Universal Robots PolyScope program: MAIN.urp

Program MAIN (installation=GD directory=/programs/GD createdIn=5.13.0 lastSavedIn=5.13.0 robotSerialNumber=20235201349)
Calibrated DH parameters: a=[0.000054, -0.419714, -0.551624, -0.000117, -0.00005, 0]; d=[0.180606, 361.576503, -382.621839, 21.219041, 0.119842, 0.115503]; alpha=[1.57022, -0.001233, 0.007049, 1.570107, -1.569424, 0]; deltaTheta=[0, -0.815667, 6.836137, 0.262718, -0.000001, 0]
InitVariablesNode
BeforeStart
  Script file /programs/GD/ROVI/ROVI_RESET.script
    | def ROVI_RESET():
    |   if (not socket_open(host,port,socket_name)):
    |     rovi_err=902
    |     return False
    |   end
    |   socket_send_line("X0()",socket_name)
    |   ret=socket_read_line(socket_name,socket_timeout)
    |   if (ret == "OK"):
    |     rovi_err=0
    |   elif (ret == "NG"):
    |     rovi_err=to_num(socket_read_line(socket_name,socket_timeout))
    |   else:
    |     ret="NG"
    |     rovi_err=903
    |   end
    |   socket_close(socket_name)
    |   if (rovi_err != 0):
    |     if (is_popup):
    |       popup(str_cat(ret,rovi_err),title="X0",warning=True,blocking=True)
    |     end
    |     return False
    |   else:
    |     return True
    |   end
    | end
  Script file /programs/GD/ROVI/ROVI_CAPTURE.script
    | def ROVI_CAPTURE():
    |   Y1=[0.0,0.0,0.0,0.0]
    | #  p=get_actual_tool_flange_pose()
    |   p=Bucket
    |   if (not socket_open(host,port,socket_name)):
    |     rovi_err=902
    |     return False
    |   end
    |   socket_send_string("X1(",socket_name)
    |   socket_send_string(p[0],socket_name)
    |   socket_send_string(",",socket_name)
    |   socket_send_string(p[1],socket_name)
    |   socket_send_string(",",socket_name)
    |   socket_send_string(p[2],socket_name)
    |   socket_send_string(",",socket_name)
    |   socket_send_string(p[3],socket_name)
    |   socket_send_string(",",socket_name)
    |   socket_send_string(p[4],socket_name)
    |   socket_send_string(",",socket_name)
    |   socket_send_string(p[5],socket_name)
    |   socket_send_line(")",socket_name)
    |   ret=socket_read_line(socket_name,socket_timeout)
    |   if (ret == "OK"):
    |     rovi_err=0
    |     f=socket_read_ascii_float(4,socket_name,socket_timeout)
    |     while (f[0]!=4):
    |       sleep(0.3)
    |       f=socket_read_ascii_float(4,socket_name,socket_timeout)
    |     end
    |     i=0
    |     while (i<4):
    |       Y1[i]=f[i+1]
    |       i=i+1
    |     end
    |   elif (ret == "NG"):
    |     rovi_err=to_num(socket_read_line(socket_name,socket_timeout))
    |   else:
    |     ret="NG"
    |     rovi_err=903
    |   end
    |   socket_close(socket_name)
    |   if (rovi_err != 0):
    |     if (is_popup):
    |       popup(str_cat(ret,rovi_err),title="X1",warning=True,blocking=True)
    |     end
    |     return False
    |   else:
    |     return True
    |   end
    | end
  Script file /programs/GD/ROVI/ROVI_SOLVE.script
    | def ROVI_SOLVE(is_popup=is_popup):
    |   buf=p[10000.0,0.0,0.0,0.0,0.0,0.0]
    |   if (not socket_open(host,port,socket_name)):
    |     rovi_err=902
    |     return False
    |   end
    |   socket_send_line("X2()",socket_name)
    |   ret=socket_read_line(socket_name,socket_timeout)
    |   if (ret == "OK"):
    |     rovi_err=0
    |     f=socket_read_ascii_float(6,socket_name,socket_timeout)
    |     while (f[0]!=6):
    |       sleep(0.3)
    |       f=socket_read_ascii_float(6,socket_name,socket_timeout)
    |     end
    |     counter=0
    |     while (counter<6):
    |       buf[counter]=f[counter+1]
    |       counter=counter+1
    |     end
    |   elif (ret == "NG"):
    |     rovi_err=to_num(socket_read_line(socket_name,socket_timeout))
    |   else:
    |     ret="NG"
    |     rovi_err=903
    |   end
    |   sleep(1.0)
    |   socket_close(socket_name)
    |   if (rovi_err != 0):
    |     if (is_popup):
    |       popup(str_cat(ret,rovi_err),title="X2",warning=True,blocking=True)
    |     end
    |   end
    |   return buf
    | end
  Script file /programs/GD/ROVI/ROVI_RECIPE.script
    | def ROVI_RECIPE(recipe):
    |   if (not socket_open(host,port,socket_name)):
    |     rovi_err=902
    |     return False
    |   end
    |   socket_send_line(str_cat(str_cat("X3(",recipe),")"),socket_name)
    |   ret=socket_read_line(socket_name,socket_timeout)
    |   if (ret == "OK"):
    |     rovi_err=0
    |   elif (ret == "NG"):
    |     rovi_err=to_num(socket_read_line(socket_name,socket_timeout))
    |   else:
    |     ret="NG"
    |     rovi_err=903
    |   end
    |   socket_close(socket_name)
    |   if (rovi_err != 0):
    |     if (is_popup):
    |       popup(str_cat(ret,rovi_err),title="X3",warning=True,blocking=True)
    |     end
    |     return False
    |   else:
    |     return True
    |   end
    | end
  Script file /programs/GD/ROVI/ROVI_PARAM.script
    | def ROVI_PARAM(prm_name,prm_value=None):
    |   Y8=0.0
    |   if (not socket_open(host,port,socket_name)):
    |     rovi_err=902
    |     return False
    |   end
    |   socket_send_string("X8(",socket_name)
    |   socket_send_string(prm_name,socket_name)
    |   if (prm_value != None):
    |     socket_send_string(" ",socket_name)
    |     socket_send_string(prm_value,socket_name)
    |   end
    |   socket_send_line(")",socket_name)
    |   ret=socket_read_line(socket_name,socket_timeout)
    |   if (ret == "OK"):
    |     rovi_err=0
    |     if (prm_value == None):  # rosparam get
    |       Y8=to_num(socket_read_line(socket_name,socket_timeout))
    |     else:    # rosparam set
    |       f=1
    |     end
    |   elif (ret == "NG"):
    |     rovi_err=to_num(socket_read_line(socket_name,socket_timeout))
    |   else:
    |     ret="NG"
    |     rovi_err=903
    |   end
    |   socket_close(socket_name)
    |   if (rovi_err != 0):
    |     if (is_popup):
    |       popup(str_cat(ret,rovi_err),title="X8",warning=True,blocking=True)
    |     end
    |     return False
    |   else:
    |     return True
    |   end
    | end
  Script file /programs/GD/CONTROL/STATUS_CONTROL.script
    | def CHECK_VT_STATUS():
    |   write_output_boolean_register(8, read_input_boolean_register(64))   # GPBO_PCOK
    |   write_output_boolean_register(9, read_input_boolean_register(65))   # GPBO_YCAMOK
    |   write_output_boolean_register(10, read_input_boolean_register(66))  # GPBO_DFOK
    |   write_output_integer_register(5, read_input_integer_register(24))   # GPIO_PayloadNo
    | end
  Script file /programs/GD/CONTROL/CYCLE_CONTROL.script
    | def GET_REG(prg_no):
    |   WorkPosNo=read_input_integer_register(4)-1                       # GPII_WorkPosNo
    |   CaptIndex[WorkPosNo]=read_input_integer_register(21)-1           # GPII_CaptColNo
    |   CaptRowNo=read_input_integer_register(20)-1        # GPII_CaptRowNo
    |   CaptStepZ=read_input_integer_register(6) / 1000.0         # GPII_CaptStepZ
    |   ReCaptNo=0
    |   if (prg_no==1203):
    |     ReCaptNo=read_input_integer_register(22)                # GPII_ReCaptNo
    |   end
    |   ReCaptZ=read_input_integer_register(7) / 1000.0         # GPII_ReCaptZ
    |   CutOffZDef=read_input_integer_register(11) / 1000.0          # GPII_CutOffZ
    |   CrankDepthFull=read_input_integer_register(10) / 1000.0   # GPII_FullDepth
    | end
    | 
    | def POSE_SUB(p, teach_frame):
    |   return pose_trans(inv(teach_frame), p)
    | end
    | 
    | def GET_BUCKET_UPPER(pos=0):
    |   if UseNewCaptPos:
    |     p=POSE_SUB(CaptPoint_C, BucketM)
    |     pX=[BKWidth/2,CaptPointL_dX,BKWidth-CaptPointR_dX]
    |     p[0]=pX[pos]
    |   else:
    |     captpos=[CaptPoint_C,CaptPoint_L,CaptPoint_R]
    |     p=captpos[pos]
    |     p=POSE_SUB(p, BucketM)
    |   end
    |   return p
    | end
    | 
    | def SET_BUCKET_DEF():
    |   BucketM=pBucketM
    |   if (WorkPosNo<0):
    |     Bucket=pBucketC
    |   else:
    |     Bucket=pBucket[WorkPosNo]
    |   end
    | end
    | 
    | def SET_BUCKET():
    |   SET_BUCKET_DEF()
    |   Bucket[2]=Bucket[2]-CaptStepZ*CaptRowNo
    | end
    | 
    | def SET_CV():
    |   CV=pCV
    | end
    | 
    | def SET_CAPT_INDEX():
    |   CaptIndexWk=CaptIndex[WorkPosNo]
    |   ReCaptZWk=0
    |   if (prg_no==1203):
    |     if   (ReCaptNo==0):
    |       if (CaptIndexWk==0):
    |         if (0<=DistPillarBak):
    |           CaptIndexWk=1
    |         else:
    |           CaptIndexWk=2
    |         end
    |         ReCaptZWk=0
    |       else:
    |         CaptIndexWk=0
    |         ReCaptZWk=0
    |       end
    |     elif (ReCaptNo==1):
    |       if (CaptIndexWk==0):
    |         CaptIndexWk=0
    |         ReCaptZWk=-ReCaptZ
    |       else:
    |         CaptIndexWk=CaptIndexWk
    |         ReCaptZWk=-ReCaptZ
    |       end
    |     else:
    |       if (CaptIndexWk==0):
    |         CaptIndexWk=0
    |         ReCaptZWk=ReCaptZ
    |       else:
    |         CaptIndexWk=CaptIndexWk
    |         ReCaptZWk=ReCaptZ
    |       end
    |     end
    |   end
    | end
    | 
    | def GET_CAPTPOS():
    |   SET_BUCKET()
    |   SET_CAPT_INDEX()
    |   if UseNewCaptPos:
    |     p=GET_BUCKET_UPPER(CaptIndexWk)
    |     p[2]=p[2]-ReCaptZWk
    |   else:
    |     captpos=[CaptPoint_C,CaptPoint_L,CaptPoint_R]
    |     p=captpos[CaptIndexWk]
    |     p[2]=p[2]-ReCaptZWk
    |     p=POSE_SUB(p, BucketM)
    |   end
    |   return p
    | end
    | 
    | def CHECK_CAPTPOS():
    |   isOK=((CaptStepZ*(read_input_integer_register(20)-1)) < (read_input_integer_register(9) / 1000.0))
    |   return isOK
    | end
    | 
    | def GET_ZSLIDE_POS(p):
    |   p[2]=p[2]-CaptStepZ*CaptRowNo
    |   return p
    | end
    | 
    | def END_CYCLE():
    |   stopl(1.2)
    |   end_force_mode()
    |   end_freedrive_mode()
    |   socket_close(socket_name)
    | end
    | 
    | def CHECK_SPEED(smax,f=[1,1,1,1,1,1]):
    |   s=TCPSpeed
    |   i=0
    |   while (i<6):
    |     if ((f[i]==1) and (smax[i]<s[i])):
    |       return False
    |     end
    |     i=i+1
    |   end
    |   return True
    | end
  Script file /programs/GD/CONTROL/ZONE_CONTROL.script
    | def GET_DIST(P1, P2):
    |   return pose_dist(P1, P2)
    | end
    | def CHECK_DIST_NEAR(P1, P2, th):
    |   return (GET_DIST(P1, P2) < th)
    | end
    | def DIST_HOME():
    |   return pose_dist(gHome_Position,CurrPos_p)
    | end
    | 
    | def CHECK_HOME():
    |   return (DIST_HOME()<ZoneDistTh)
    | end
    | 
    | def GET_DEST_FLANGE(target, feature, tcp):
    |   return pose_trans(pose_trans(feature, target), pose_inv(tcp))
    | end
    | 
    | def DIST_CVFront():
    |   if (read_input_integer_register(4)==1):
    |     p=g2GD_pos1
    |   else:
    |     p=g1GD_pos1
    |   end
    |   return pose_dist(p,CurrPos_p)
    | end
    | 
    | def CHECK_CVFront():
    |   return (DIST_CVFront()<ZoneDistTh)
    | end
    | 
    | def CHECK_RB_POS(prg_no):
    |   ret=True
    |   if (prg_no==1001):
    |     ret=CHECK_ALLOW_GO_HOME(0)
    |   end
    |   if ((prg_no==1201) or (prg_no==1401) or (prg_no==1402) or (prg_no==6001) or (prg_no==6101) or (prg_no==6401) or (prg_no==6102) or (prg_no==7001)):
    |     ret=CHECK_HOME()
    |   end
    |   if ((prg_no==1002) or (prg_no==1241) or (prg_no==1261)):
    |     ret=CHECK_BKInside()
    |   end
    |   if (prg_no==1251):
    |     ret=(CHECK_HOME() or CHECK_CVUpper())
    |   end
    |   if (ret != True):
    |     SubPrgResult=801
    |     sleep(999999.0)
    |   end
    | end
    | 
    | def DIST_ORIGIN():
    |   p=CurrPos_p
    |   o=p
    |   o[0]=0.0
    |   o[1]=0.0
    |   DistOrigin=pose_dist(o,p)
    |   return pose_dist(o,p)
    | end
    | 
    | def CHECK_EVAC_ORG():
    |   return (EvacRadiusTh<DIST_ORIGIN())
    | end
    | 
    | def CHECK_EVAC_X():
    |   return (EvacXTh[0]<CurrPos_p[0] and CurrPos_p[0]<EvacXTh[1])
    | end
    | 
    | def CHECK_EVAC_Y():
    |   return (EvacYTh[0]<CurrPos_p[1] and CurrPos_p[1]<EvacYTh[1])
    | end
    | 
    | def CHECK_EVAC_Z():
    |   return (EvacZTh[0]<CurrPos_p[2] and CurrPos_p[2]<EvacZTh[1])
    | end
    | 
    | def CHECK_EVAC():
    |   ret=True
    |   ret=(ret and CHECK_EVAC_ORG())
    |   ret=(ret and CHECK_EVAC_X())
    |   ret=(ret and CHECK_EVAC_Y())
    |   ret=(ret and CHECK_EVAC_Z())
    |   return ret
    | end
    | 
    | def CHECK_BKInside():
    |   ret=True
    |   pos=read_input_integer_register(4)
    |   if (pos>2):
    |     ret=False
    |   else:
    |     if (not read_input_boolean_register(13+pos)):
    |       ret=False
    |       ver_3=read_input_boolean_register(13+pos)
    |     else:
    |       bk=pBucket[pos-1]
    |       if (pos==1):
    |         ret=(ret and CurrPos_p[0]>ZoneHomeX)
    |         ret=(ret and bk[1]-(BucketWidth-ZoneBucketGap)<CurrPos_p[1] and CurrPos_p[1]<bk[1]-ZoneBucketGap)
    |       elif (pos==2):
    |         ret=(ret and CurrPos_p[0]<-ZoneHomeX)
    |         ret=(ret and bk[1]+ZoneBucketGap<CurrPos_p[1] and CurrPos_p[1]<bk[1]+(BucketWidth-ZoneBucketGap))
    |       end
    |     end
    |   end
    |   return ret
    | end
    | 
    | def CHECK_CVOutside():
    |   ret=True
    |   ret=(ret and gCV_11_M[0]-Zone6ThX<CurrPos_p[0])
    |   ret=(ret and CurrPos_p[0]<gCV_11_M[0]+Zone6ThX)
    |   ret=(ret and gCV_11_M[1]-Zone6ThY<CurrPos_p[1])
    |   ret=(ret and CurrPos_p[1]<gCV_11_M[1]+Zone6ThY)
    |   return (not ret)
    | end
    | 
    | def CHECK_CVUpper():
    |   ret=True
    |   ret=(ret and (CVXTh[0]<CurrPos_p[0] and CurrPos_p[0]<CVXTh[1]))
    |   ret=(ret and (CVYTh[0]<CurrPos_p[1] and CurrPos_p[1]<CVYTh[1]))
    |   ret=(ret and (CVZTh[0]<CurrPos_p[2] and CurrPos_p[2]<CVZTh[1]))
    |   return ret
    | end
    | 
    | def CHECK_ALLOW_GO_HOME(no=0):
    |   ret=False
    |   if (no==0 or no==1):
    |     ret=(ret or CHECK_EVAC())
    |     v1=ret
    |   end
    |   if (no==0 or no==2):
    |     ret=(ret or CHECK_BKInside())
    |     v2=ret
    |   end
    |   if (no==0 or no==3):
    |     ret=(ret or CHECK_CVUpper())
    |     v3=ret
    |   end
    |   return ret
    | end
    | 
    | def CHECK_ZONE(no):
    |   if (no==1):
    |     return (CurrPos_p[2]>=Zone1ZTh)
    |   elif (no==2):
    |     return (CurrPos_p[0]>ZoneHomeX)
    |   elif (no==3):
    |     return (CurrPos_p[0]<-ZoneHomeX)
    |   elif (no==4):
    |     return CHECK_CVFront()
    |   elif (no==5):
    |     return CHECK_BKInside()
    |   elif (no==6):
    |     return CHECK_CVOutside()
    |   elif (no==7):
    |     return CHECK_CVUpper()
    |   end
    | end
  Script file /programs/GD/CONTROL/ALIGN_AXIS.script
    | def GET_NORM_VEC(p,axis=2):
    |   rot=p[0.0, 0.0, 0.0, p[3], p[4], p[5]]
    |   vec=p[0.0, 0.0, 0.0, 0.0, 0.0, 0.0]
    |   vec[axis]=1.0
    |   norm_p=pose_trans(rot,vec)
    |   return [norm_p[0], norm_p[1], norm_p[2]]
    | end
    | 
    | def GET_INNER_PRODUCT(v1,v2):
    |   return v1[0]*v2[0]+v1[1]*v2[1]+v1[2]*v2[2]
    | end
    | def GET_OUTER_PRODUCT(v1,v2):
    |   x=v1[1]*v2[2]-v1[2]*v2[1]
    |   y=v1[2]*v2[0]-v1[0]*v2[2]
    |   z=v1[0]*v2[1]-v1[1]*v2[0]
    |   return [x,y,z]
    | end
    | def GET_THETA(v1,v2):
    | #  cos=GET_INNER_PRODUCT(v1,v2) / norm(v1) / norm(v2)
    |   cos=GET_INNER_PRODUCT(v1,v2)
    |   g_cos=cos
    |   theta=norm(acos(cos))
    |   return theta
    | end
    | 
    | def GET_ALIGNED_POSE(target,feature,axis=2):
    |   feature_from_target=pose_trans(pose_inv(target),feature)
    |   g_f_from_t=feature_from_target
    |   nz_feature_from_target=GET_NORM_VEC(feature_from_target,axis)
    |   g_nz_f_from_t=nz_feature_from_target
    |   nz_target_from_target=[0.0, 0.0, 0.0]
    |   nz_target_from_target[axis]=1.0
    |   g_nz_t_from_t=nz_target_from_target
    | 
    |   theta=GET_THETA(nz_feature_from_target,nz_target_from_target)
    |   g_theta=theta
    |   rot_vec_n=normalize(GET_OUTER_PRODUCT(nz_target_from_target,nz_feature_from_target))
    | 
    |   if theta>d2r(90.0):
    |     theta=theta-d2r(180.0)
    |   end
    |   rot_vec=rot_vec_n * (theta)
    |   rot_p=p[0.0,0.0,0.0,rot_vec[0],rot_vec[1],rot_vec[2]]
    |   return pose_trans(target,rot_p)
    | end
    | def GET_ALIGNED_TCP(feature,axis=2):
    |   tcp=get_actual_tcp_pose()
    |   return GET_ALIGNED_POSE(tcp,feature,axis)
    | end
  Script file /programs/GD/CONTROL/ROTATE_CONTROL.script
    | def GET_TCP_FORCE_TOOL():
    |   force_torque=get_tcp_force()
    |   force_B=p[force_torque[0], force_torque[1], force_torque[2], 0, 0, 0]
    |   torque_B=p[force_torque[3], force_torque[4], force_torque[5], 0, 0, 0]
    |   tcp=get_actual_tcp_pose()
    |   rotation_BT=p[0, 0, 0, tcp[3], tcp[4], tcp[5]]
    |   force_T=pose_trans(pose_inv(rotation_BT), force_B)
    |   torque_T=pose_trans(pose_inv(rotation_BT), torque_B)
    |   force_torque_T=p[force_T[0], force_T[1], force_T[2], torque_T[0], torque_T[1], torque_T[2]]
    |   return force_torque_T
    | end
    | 
    | def CHECK_VALUE_RZ():
    |   return True
    | end
    | 
    | def GET_FORCE_VALUE_RZ(target):
    |   PoseSub= pose_sub (CurrPos_p,target)
    |   RYSub=r2d(PoseSub[4])
    |   RZSub=r2d(PoseSub[5])
    | #  if (RYSub<RZSupRYRange[0] or RZSupRYRange[1]<RYSub):
    | #    RZSupForceVal=0.0
    | #    return RZSupForceVal
    | #  end
    |   if (RZSub<0):
    |     RZMin=RZSupDegMin[0]
    |     RZRatio=RZSupRatio[0]
    |     RZOffset=RZSupOffset[0]
    |   else:
    |     RZMin=RZSupDegMin[1]
    |     RZRatio=RZSupRatio[1]
    |     RZOffset=-RZSupOffset[1]
    |   end
    |   if (norm(RZSub) >= norm(RZMin)):
    |     RZSupForceVal=(RZMin-RZSub)*RZRatio+RZOffset
    |   else:
    |     RZSupForceVal=0
    |   end
    |   if (RZSupForceVal<RZSupForceRange[0]):
    |     RZSupForceVal=RZSupForceRange[0]
    |   elif (RZSupForceRange[1]<RZSupForceVal):
    |     RZSupForceVal=RZSupForceRange[1]
    |   end
    |   if (RYSub<RZSupRYRange[0] or RZSupRYRange[1]<RYSub):
    |     RZSupForceVal=0
    |   end
    |   if ((not UseRZSupStep1) and (ForceStep==1)):
    |     RZSupForceVal=0
    |   end
    |   return RZSupForceVal
    | end
    | 
    | def GET_CVCORR_VALUE(target):
    |   CVCorrYVal=0
    |   CVCorrRZVal=0
    |   if (UseCVCorr and (not UseCVCorrCam)):
    |     PoseSub=pose_sub(CurrPos_p,target)
    |     RYSub=r2d(PoseSub[4])
    |     CVCorrRYSub=RYSub
    |     if (RYSub<0):
    |       RYMin=-CVCorrDegMin[0]
    |       RZRatio=CVCorrRatio[0]
    |       RZOffset=-CVCorrOffset[0]
    |     else:
    |       RYMin=-CVCorrDegMin[1]
    |       RZRatio=CVCorrRatio[1]
    |       RZOffset=CVCorrOffset[1]
    |     end
    |     if (norm(RYSub) >= norm(RYMin)):
    |       t=get_tcp_offset()
    |       CVCorrYVal=-t[2]*sin(d2r(RYSub))
    |       CVCorrRZVal=RYSub*RZRatio+RZOffset
    |     else:
    |       CVCorrYVal=0
    |       CVCorrRZVal=0
    |     end
    |   end
    | end
    | 
    | def GET_CVCORR_POS(target):
    |   if UseCVCorr:
    |     if (not UseCVCorrCam):
    |       pos= pose_add (p[0,0,0,0,0,d2r(-CVCorrRZVal)],p[0,0,0,target[3],target[4],target[5]])
    |       pos=p[target[0],target[1],target[2],pos[3],pos[4],pos[5]]
    |     else:
    |       pos=target
    |     end
    |   else:
    |     pos=target
    |   end
    |   return pos
    | end
    | 
    | def CHECK_RX_TILT(target):
    |   PosSub=pose_sub(CurrPos_p,target)
    |   RXSub=r2d(PoseSub[3])
    |   return (RXTiltDegMin[0]<RXSub and RXSub<RXTiltDegMin[1])
    | end
  SuppressedNode
    Script file /programs/GD/CONTROL/LOG.script
      | def POPUP_CAPT_OPTION():
      |   msg=""
      |   msg=str_cat(msg,str_cat(CaptIndex[WorkPosNo],","))
      |   msg=str_cat(msg,str_cat(ReCaptZ,","))
      |   msg=str_cat(msg,str_cat(prg_no,","))
      |   msg=str_cat(msg,str_cat(DistPillarBak,","))
      |   msg=str_cat(msg,str_cat(ReCaptNo,","))
      |   msg=str_cat(msg,str_cat(CaptIndexWk,","))
      |   msg=str_cat(msg,str_cat(ReCaptZWk,","))
      |   msg=str_cat(msg,str_cat(read_output_integer_register(2),","))
      |   msg=str_cat(msg,str_cat(WorkPosNo,","))
      |   msg=str_cat(msg,str_cat(CaptRowNo,","))
      |   popup(msg,title="CAPT_OPTION",warning=True,blocking=True)
      | end
  Script file /programs/GD/THREAD/THREAD_ROVI.script
    | thread THREAD_ROVI():
    |   THREAD_ROVI_FLG=0
    |   THREAD_ROVI_ERR=0
    |   if ((THREAD_ROVI_ERR==0) and (not ROVI_RECIPE(read_input_integer_register(2)+WorkNoOffset))):
    |     THREAD_ROVI_ERR=rovi_err
    |   end
    |   if ((THREAD_ROVI_ERR==0) and (not ROVI_RESET())):
    |     THREAD_ROVI_ERR=rovi_err
    |   end
    |   if ((THREAD_ROVI_ERR==0) and (not  ROVI_CAPTURE())):
    |     THREAD_ROVI_ERR=rovi_err
    |   end
    |   if (THREAD_ROVI_ERR==0):
    |     global Y2=ROVI_SOLVE()
    |     if ((Y2[0] == 10000.)):
    |       THREAD_ROVI_ERR=rovi_err
    |     end
    |   end
    |   THREAD_ROVI_FLG=1
    | end
    | def RUN_THREAD_ROVI():
    |   return run THREAD_ROVI()
    | end
    | def JOIN_THREAD_ROVI(thrd):
    |   if (thrd>0):
    |     join thrd
    |   end
    | end
    | def RESET_THREAD_ROVI():
    |   THREAD_ROVI_FLG=2
    |   THREAD_ROVI_ERR=-1
    | end
    | def KILL_THREAD_ROVI(thrd):
    |   if (THREAD_ROVI_FLG==0):
    |     kill thrd
    |   end
    | end
Robot Program (runOnlyOnce=false)
  Script: position_deviation_warning(True,0.4)
  Folder PREPARE_PICK_TCP
    Set NoAction tcp=TCP_RX
    PickTCP := get_tcp_offset()
  SetPayload (workpieceName=k10)
  Set NoAction tcp=TCP_1
  CutOffTCP := get_tcp_offset()
  Script: RESET_THREAD_ROVI()
  thrd108 := 0
  Set ExpressionOutput pin=GPIO_PrgNo; expression=0
  Set DigitalOutput pin=GPBO_PrgBegin; digitalValue=0
  Set DigitalOutput pin=GPBO_PrgEnd; digitalValue=0
  Set DigitalOutput pin=GPBO_PrgRun; digitalValue=0
  Set DigitalOutput pin=GPBO_BKPosDone; digitalValue=0
  Set DigitalOutput pin=GPBO_BLStop; digitalValue=0
  Set DigitalOutput pin=GPBO_BLStart; digitalValue=0
  Set DigitalOutput pin=GPBO_Released; digitalValue=0
  Wait DigitalInput pin=GPBI_PrgStart; digitalValue=0
  Wait DigitalInput pin=GPBI_PrgStart; digitalValue=1
  Set ExpressionOutput pin=GPIO_PrgResult; expression=0
  prg_no := GPII_PrgNo
  If ( not GPBI_PrgStop≠ False ) (checkContinuously=true)
    Script: CHECK_RB_POS(prg_no)
    Set ExpressionOutput pin=GPIO_PrgNo; expression=prg_no
    Wait Sleep waitTime=0.1
    Set SingleDigitalPulseActionState SingleDigitalPulseActionState(hiPulseInSeconds=1, pin=GP_bool_out[4])
    SubPrgResult := 100
    If (SubPrgResult≟100) (checkContinuously=true)
      Script: GET_REG(prg_no)
      Switch expression=prg_no
        Case (caseValue=1001)
          Script: CHECK_RB_POS(prg_no)
          Set ExpressionOutput pin=GPIO_SubPrgNo; expression=109
          Call SUB_109
          Set ExpressionOutput pin=GPIO_SubPrgNo; expression=003
          Call SUB_003
        SuppressedNode
          Case (caseValue=1002)
            Set ExpressionOutput pin=GPIO_SubPrgNo; expression=102
            Call SUB_002
            Set ExpressionOutput pin=GPIO_SubPrgNo; expression=001
            Call SUB_003
        Case (caseValue=1201)
          Set ExpressionOutput pin=GPIO_SubPrgNo; expression=101
          Call SUB_101
          Set ExpressionOutput pin=GPIO_SubPrgNo; expression=102
          Call SUB_102
          Set ExpressionOutput pin=GPIO_SubPrgNo; expression=104
          SuppressedNode
            Call SUB_104
          SuppressedNode
            Call SUB_104RX
          SuppressedNode
            Call SUB_104RXF
          Call SUB_104RXFF
          Set ExpressionOutput pin=GPIO_SubPrgNo; expression=105
          Call SUB_105
          Set ExpressionOutput pin=GPIO_SubPrgNo; expression=106
          Call SUB_106
          Set ExpressionOutput pin=GPIO_SubPrgNo; expression=108
          Call SUB_108
          Set ExpressionOutput pin=GPIO_SubPrgNo; expression=121
          Call SUB_121
          Set ExpressionOutput pin=GPIO_SubPrgNo; expression=122
          Call SUB_122
          Set ExpressionOutput pin=GPIO_SubPrgNo; expression=001
          Call SUB_001
          If (CandCnt≟1)
            SubPrgResult := 990
            Wait Sleep waitTime=999999
        Case (caseValue=1202)
          Set ExpressionOutput pin=GPIO_SubPrgNo; expression=102
          Call SUB_102
          Set ExpressionOutput pin=GPIO_SubPrgNo; expression=104
          SuppressedNode
            Set ExpressionOutput pin=GPIO_SubPrgNo; expression=104
          SuppressedNode
            Call SUB_104
          SuppressedNode
            Call SUB_104RX
          SuppressedNode
            Call SUB_104RXF
          Call SUB_104RXFF
          Set ExpressionOutput pin=GPIO_SubPrgNo; expression=105
          Call SUB_105
          Set ExpressionOutput pin=GPIO_SubPrgNo; expression=106
          Call SUB_106
          Set ExpressionOutput pin=GPIO_SubPrgNo; expression=108
          Call SUB_108
          Set ExpressionOutput pin=GPIO_SubPrgNo; expression=121
          Call SUB_121
          Set ExpressionOutput pin=GPIO_SubPrgNo; expression=122
          Call SUB_122
          Set ExpressionOutput pin=GPIO_SubPrgNo; expression=001
          Call SUB_001
          If (CandCnt≟1)
            SubPrgResult := 990
            Wait Sleep waitTime=999999
        Case (caseValue=1203)
          Set ExpressionOutput pin=GPIO_SubPrgNo; expression=103
          Call SUB_103
          Set ExpressionOutput pin=GPIO_SubPrgNo; expression=104
          SuppressedNode
            Call SUB_104
          SuppressedNode
            Call SUB_104RX
          SuppressedNode
            Call SUB_104RXF
          Call SUB_104RXFF
          Set ExpressionOutput pin=GPIO_SubPrgNo; expression=105
          Call SUB_105
          Set ExpressionOutput pin=GPIO_SubPrgNo; expression=106
          Call SUB_106
          Set ExpressionOutput pin=GPIO_SubPrgNo; expression=108
          Call SUB_108
          Set ExpressionOutput pin=GPIO_SubPrgNo; expression=121
          Call SUB_121
          Set ExpressionOutput pin=GPIO_SubPrgNo; expression=122
          Call SUB_122
          Set ExpressionOutput pin=GPIO_SubPrgNo; expression=001
          Call SUB_001
          If (CandCnt≟1)
            SubPrgResult := 990
            Wait Sleep waitTime=999999
        Case (caseValue=1241)
          Set ExpressionOutput pin=GPIO_SubPrgNo; expression=107
          Call SUB_107
          Set ExpressionOutput pin=GPIO_SubPrgNo; expression=106
          Call SUB_106
          Set ExpressionOutput pin=GPIO_SubPrgNo; expression=108
          Call SUB_108
          Set ExpressionOutput pin=GPIO_SubPrgNo; expression=121
          Call SUB_121
          Set ExpressionOutput pin=GPIO_SubPrgNo; expression=122
          Call SUB_122
          Set ExpressionOutput pin=GPIO_SubPrgNo; expression=001
          Call SUB_001
        Case (caseValue=1251)
          Set ExpressionOutput pin=GPIO_SubPrgNo; expression=107
          Call SUB_107
          Set ExpressionOutput pin=GPIO_SubPrgNo; expression=120
          Call SUB_120
          Set ExpressionOutput pin=GPIO_SubPrgNo; expression=108
          Call SUB_108
          Set ExpressionOutput pin=GPIO_SubPrgNo; expression=121
          Call SUB_121
          Set ExpressionOutput pin=GPIO_SubPrgNo; expression=122
          Call SUB_122
          Set ExpressionOutput pin=GPIO_SubPrgNo; expression=001
          Call SUB_001
        Case (caseValue=1261)
          Set ExpressionOutput pin=GPIO_SubPrgNo; expression=161
          Call SUB_161
          Set ExpressionOutput pin=GPIO_SubPrgNo; expression=001
          Call SUB_001
        Case (caseValue=1281)
          Set ExpressionOutput pin=GPIO_SubPrgNo; expression=181
          Call SUB_181
          Set ExpressionOutput pin=GPIO_SubPrgNo; expression=001
          Call SUB_001
        Case (caseValue=1401)
          Set ExpressionOutput pin=GPIO_SubPrgNo; expression=141
          Call SUB_141
          Script: pBucket[WorkPosNo]=Y2
          Set ExpressionOutput pin=GPIO_SubPrgNo; expression=143
          Call SUB_143
          Set SingleDigitalPulseActionState SingleDigitalPulseActionState(hiPulseInSeconds=1, pin=GP_bool_out[13])
        Case (caseValue=1402)
          Set ExpressionOutput pin=GPIO_SubPrgNo; expression=142
          Call SUB_142
          Set ExpressionOutput pin=GPIO_SubPrgNo; expression=001
          Call SUB_001
          Script: pCV=Y2
        Case (caseValue=3100)
          Set ExpressionOutput pin=GPIO_SubPrgNo; expression=3100
          Call SUB_3100
        Case (caseValue=6001)
          Set ExpressionOutput pin=GPIO_SubPrgNo; expression=6001
          Call SUB_6001
        Case (caseValue=6101)
          CheckMST := 0
          Set ExpressionOutput pin=GPIO_SubPrgNo; expression=6101
          Call SUB_6101
        Case (caseValue=6102)
          If (GPII_CheckMST>0)
            CheckMST := GPII_CheckMST
            WorkPosNo := -1
            CaptRowNo := 5
            SuppressedNode
              CaptRowNo := 3
            Script: SET_BUCKET()
            Set ExpressionOutput pin=GPIO_SubPrgNo; expression=6101
            Call SUB_6101
          Set ExpressionOutput pin=GPIO_SubPrgNo; expression=6102
          SuppressedNode
            Call SUB_6102
          SuppressedNode
            Call SUB_6102RX
          SuppressedNode
            Call SUB_6102RXF
          Call SUB_6102RXFF
        Case (caseValue=6401)
          Set ExpressionOutput pin=GPIO_SubPrgNo; expression=141
          Call SUB_141
          Script: pBucketM=Y2
          Script: pBucket[WorkPosNo]=Y2
        Case (caseValue=6402)
          Set ExpressionOutput pin=GPIO_SubPrgNo; expression=142
          Call SUB_6402
        Case (caseValue=7001)
          Set ExpressionOutput pin=GPIO_SubPrgNo; expression=7001
          Call SUB_7001
        Case (caseValue=7002)
          Set ExpressionOutput pin=GPIO_SubPrgNo; expression=7002
          Call SUB_7002
    Set ExpressionOutput pin=GPIO_PrgResult; expression=SubPrgResult
  Script: END_CYCLE()
  If GPBI_PrgStop≟ True
    SubPrgResult := 800
    Set ExpressionOutput pin=GPIO_PrgResult; expression=SubPrgResult
    Set ExpressionOutput pin=GPBO_PrgRun; expression=False
  Wait Sleep waitTime=0.1
  prg_no := 0
  SetPayload (workpieceName=k10)
  Set NoAction tcp=TCP_1
  If (GPIO_PrgNo≠0)
    Set SingleDigitalPulseActionState SingleDigitalPulseActionState(hiPulseInSeconds=1, pin=GP_bool_out[5])
    Set ExpressionOutput pin=GPIO_PrgNo; expression=0
  Wait DigitalInput pin=GPBI_PrgStart; digitalValue=0
  Wait DigitalInput pin=GPBI_PrgStop; digitalValue=0
Thread スレッド_2 (runOnlyOnce=false)
  Sub3100_GPII18 := GPII_RunOption
  Script: CurrPos=get_actual_tool_flange_pose()
  Script: CurrPos_p=get_actual_tcp_pose()
  Script: Currpos_p_UF0=pose_trans(pose_inv(UF), CurrPos_p)
  TCPSpeed := get_actual_tcp_speed()
  TCPForce := get_tcp_force()
  TCPForceTL := GET_TCP_FORCE_TOOL()
  Set ExpressionOutput pin=GPBO_RBHome; expression=CHECK_HOME()
  Set ExpressionOutput pin=GPBO_AllowGoHom; expression=CHECK_ALLOW_GO_HOME(0)
  Set ExpressionOutput pin=GPBO_Zone01; expression=CHECK_ZONE(1)
  Set ExpressionOutput pin=GPBO_Zone02; expression=CHECK_ZONE(2)
  Set ExpressionOutput pin=GPBO_Zone03; expression=CHECK_ZONE(3)
  Set ExpressionOutput pin=GPBO_Zone04; expression=CHECK_ZONE(4)
  Set ExpressionOutput pin=GPBO_Zone05; expression=CHECK_ZONE(5)
  Set ExpressionOutput pin=GPBO_Zone06; expression=CHECK_ZONE(6)
  Set ExpressionOutput pin=GPBO_Zone07; expression=CHECK_ZONE(7)
  Set ExpressionOutput pin=GP_bool_out[31]; expression=CHECK_ALLOW_GO_HOME(1)
  Script: CHECK_VT_STATUS()
  Script: sync()
SubProgram  [hidden by the author, left out]
SuppressedNode
  SubProgram  [hidden by the author, left out]
SubProgram -> SUB_003
SubProgram -> SUB_101
SubProgram -> SUB_102
SubProgram  [hidden by the author, left out]
SuppressedNode
  SubProgram  [hidden by the author, left out]
SuppressedNode
  SubProgram  [hidden by the author, left out]
SuppressedNode
  SubProgram  [hidden by the author, left out]
SubProgram -> SUB_104RXFF
SubProgram -> SUB_105
SubProgram -> SUB_106
SubProgram -> SUB_107
SubProgram -> SUB_108
SubProgram -> SUB_109
SubProgram -> SUB_120
SubProgram -> SUB_121
SubProgram -> SUB_122
SubProgram -> SUB_141
SubProgram -> SUB_142
SubProgram -> SUB_143
SubProgram  [hidden by the author, left out]
SubProgram  [hidden by the author, left out]
SubProgram -> SUB_3100
SubProgram -> SUB_6001
SubProgram -> SUB_6101
SuppressedNode
  SubProgram  [hidden by the author, left out]
SuppressedNode
  SubProgram  [hidden by the author, left out]
SuppressedNode
  SubProgram  [hidden by the author, left out]
SubProgram -> SUB_6102RXFF
SubProgram -> SUB_6402
SubProgram  [hidden by the author, left out]
SubProgram  [hidden by the author, left out]
SubProgram SUB_109 (keepSynchronizedWithDisk=true) programFile=/programs/GD/SUB_109.urp
  If CHECK_ALLOW_GO_HOME(2) or CHECK_ALLOW_GO_HOME(3)
    If GPBI_WorkExists and GPBI_BLLoad0
      Set NoAction tcp=TCP_RXF
      SetPayload (workpieceName=k2)
      Folder ROVI_RECIPE
        If (not ROVI_RECIPE(GPII_WorkNo+WorkNoTL))
          SubPrgResult := rovi_err
          Wait Sleep waitTime=999999
      Folder ROVI_RESET
        If (not ROVI_RESET())
          SubPrgResult := rovi_err
          Wait Sleep waitTime=999999
      Set SingleDigitalPulseActionState SingleDigitalPulseActionState(hiPulseInSeconds=1, pin=GP_bool_out[14])
      Folder ROVI_CAPTURE
        Script: force_mode_set_damping(0)
        Script: force_mode_set_gain_scaling(0.5)
        Wait Sleep waitTime=0.02
        Script: zero_ftsensor()
        Force Frame feature=Joint_6_name; selection=[0, 0, 0, 1, 0, 0]; wrench=[0, 30, 0, 5, 10, 0]; limitsForce=[0.15, 0.03, 0.01, 0.087266, 0.087266, 1.047198]; limitsMotion=[0.1, 0.1, 0.1, 0.349066, 0.349066, 0.349066]
          forceON := True
          Loop While (checkContinuously=false) expression=forceON
            If TCPForceTL[3]<-2 (checkContinuously=true)
              Wait Sleep waitTime=1
              forceON := False
            Wait Sleep waitTime=0.1
        Wait Sleep waitTime=3
        Script: force_mode_set_gain_scaling(1)
        Script: force_mode_set_damping(0)
        If ( not ROVI_CAPTURE())
          SubPrgResult := rovi_err
          Wait Sleep waitTime=999999
      Folder ROVI_SOLVE
        Y2 := ROVI_SOLVE()
        If (Y2[0]≟10000.)
          SubPrgResult := rovi_err
          Wait Sleep waitTime=999999
      SetPayload (workpieceName=k10)
      UF := Y2
      MoveL speed 200 mm/s, acceleration 70 mm/s^2 (useActiveTCP=false) tcp=TCP_1; feature=UF
        Wait Sleep waitTime=1
        Waypoint Variable (Variable): variable(featureName=gCV_11_M)
        Waypoint Variable (Variable): variable(featureName=gCV_12_M)
      MoveL speed 200 mm/s, acceleration 70 mm/s^2 (useActiveTCP=false) tcp=TCP_1; feature=UF
        Waypoint Variable (Variable): motionParameters(jointSpeed=1.047198 jointAcceleration=1.396263 cartesianSpeed=0.03 cartesianAcceleration=0.03); variable(featureName=gCV_13_M)
        Waypoint Variable (Variable): variable(featureName=gCV_14_M)
      Set SingleDigitalPulseActionState SingleDigitalPulseActionState(hiPulseInSeconds=1, pin=GP_bool_out[15])
SubProgram SUB_003 (keepSynchronizedWithDisk=true) programFile=/programs/GD/SUB_003.urp
  If CHECK_ALLOW_GO_HOME(3)
    If GPBI_WorkExists and GPBI_BLLoad1 and ( not GPBI_BLLoad0) (checkContinuously=true)
      SetPayload (workpieceName=k120)
      MoveL speed 250 mm/s, acceleration 50 mm/s^2 (useActiveTCP=true) feature=CV
        Waypoint Variable (Variable): variable(featureName=gCV_2_M)
      SetPayload (workpieceName=k10)
      MoveL speed 400 mm/s, acceleration 140 mm/s^2 (useActiveTCP=true) feature=CV
        Waypoint Variable (Variable): variable(featureName=g1GD_pos2)
      MoveJ speed 70 deg/s, acceleration 30 deg/s^2 (useActiveTCP=false) tcp=TCP_1; feature=Base
        Waypoint Variable (Variable): variable(featureName=gHome_Position)
    ElseIf ( not GPBI_WorkExists) and ( not GPBI_BLLoad1) and GPBI_BLLoad0
      SetPayload (workpieceName=k10)
      MoveL speed 250 mm/s, acceleration 50 mm/s^2 (useActiveTCP=true) feature=CV
        Waypoint Variable (Variable): variable(featureName=gCV_13_M)
        Waypoint Variable (Variable): variable(featureName=gCV_14_M)
      MoveL speed 400 mm/s, acceleration 140 mm/s^2 (useActiveTCP=true) feature=CV
        Waypoint Variable (Variable): variable(featureName=g1GD_pos2)
      MoveJ speed 70 deg/s, acceleration 30 deg/s^2 (useActiveTCP=false) tcp=TCP_1; feature=Base
        Waypoint Variable (Variable): variable(featureName=gHome_Position)
  ElseIf CHECK_ALLOW_GO_HOME(2)
    SetPayload (workpieceName=k120)
    Script: sync()
    If (WorkPosNo≟0)
      MoveL speed 250 mm/s, acceleration 50 mm/s^2 (useActiveTCP=true) feature=Base
        Waypoint Variable (Variable): variable(featureName=g2GD_pos5)
      MoveL speed 400 mm/s, acceleration 140 mm/s^2 (useActiveTCP=true) feature=Base
        SetPayload (workpieceName=k10)
        SuppressedNode
          Waypoint Variable (Variable): variable(featureName=g2GD_pos4)
        Waypoint Variable (Variable): motionParameters(blendRadius=0.1); variable(featureName=g2GD_pos3)
        Waypoint Variable (Variable): motionParameters(jointSpeed=1.047198 jointAcceleration=1.396263 cartesianSpeed=0.4 cartesianAcceleration=0.07); variable(featureName=g2GD_pos2)
    ElseIf (WorkPosNo≟1)
      MoveL speed 250 mm/s, acceleration 50 mm/s^2 (useActiveTCP=true) feature=Base
        Waypoint Variable (Variable): variable(featureName=g1GD_pos5)
      MoveL speed 400 mm/s, acceleration 140 mm/s^2 (useActiveTCP=true) feature=Base
        SetPayload (workpieceName=k10)
        Waypoint Variable (Variable): variable(featureName=g1GD_pos3)
        Waypoint Variable (Variable): variable(featureName=g1GD_pos2)
    MoveJ speed 70 deg/s, acceleration 30 deg/s^2 (useActiveTCP=false) tcp=TCP_1; feature=Base
      Waypoint Variable (Variable): variable(featureName=gHome_Position)
  ElseIf CHECK_ALLOW_GO_HOME(1)
    SetPayload (workpieceName=k10)
    MoveJ speed 70 deg/s, acceleration 30 deg/s^2 (useActiveTCP=false) tcp=TCP_1; feature=Base
      Waypoint Variable (Variable): variable(featureName=gHome_Position)
  Set NoAction tcp=TCP_1
SubProgram SUB_002 [hidden by the author, left out]
SubProgram SUB_101 (keepSynchronizedWithDisk=true) programFile=/programs/GD/SUB_101.urp
  Folder INITIALIZE
    SetPayload (workpieceName=k10)
  Folder BUCKET
    Script: SET_BUCKET_DEF()
    BucketUpperPos := GET_BUCKET_UPPER()
  MoveJ speed 40 deg/s, acceleration 20 deg/s^2 (useActiveTCP=false) tcp=TCP_1; feature=Bucket
    Waypoint Variable (Variable): variable=BucketUpperPos
SubProgram SUB_102 (keepSynchronizedWithDisk=true) programFile=/programs/GD/SUB_102.urp
  Folder ROVI_RECIPE
    If (not ROVI_RECIPE(GPII_WorkNo))
      SubPrgResult := rovi_err
      Wait Sleep waitTime=999999
  Folder ROVI_PARAM
    If ( not ROVI_PARAM(BKWidth_Name,BKWidth_Value[WorkPosNo]))
      SubPrgResult := rovi_err
      Wait Sleep waitTime=999999
  Folder ROVI_RESET
    If (not ROVI_RESET())
      SubPrgResult := rovi_err
      Wait Sleep waitTime=999999
  SetPayload (workpieceName=k120)
  Folder ROVI_CAPTURE
    If ( not CHECK_CAPTPOS())
      SubPrgResult := 802
      Wait Sleep waitTime=999999
    SetPayload (workpieceName=k120)
    CaptPos := GET_CAPTPOS()
    MoveJ speed 40 deg/s, acceleration 20 deg/s^2 (useActiveTCP=false) tcp=TCP_1; feature=Bucket
      Waypoint Variable (Variable): variable=CaptPos
    Wait Sleep waitTime=1
    SuppressedNode
      Script: POPUP_CAPT_OPTION()
SubProgram SUB_104 [hidden by the author, left out]
SubProgram SUB_104RX [hidden by the author, left out]
SubProgram SUB_104RXF [hidden by the author, left out]
SubProgram SUB_104RXFF (keepSynchronizedWithDisk=true) programFile=/programs/GD/SUB_104RXFF.urp
  Script: SET_BUCKET()
  Folder ROVI_CAPTURE
    If ( not ROVI_CAPTURE())
      SubPrgResult := rovi_err
      Wait Sleep waitTime=999999
    CandCnt := Y1[0]
    DistPillar := Y1[1] / 1000.0
    LevelZ := Y1[2] / 1000.0
    NeighborZ := Y1[3] / 1000.0
    If (GPII_PrgNo≠1203)
      DistPillarBak := DistPillar
    If (CandCnt<1)
      SubPrgResult := 990
      Wait Sleep waitTime=999999
  Folder ROVI_SOLVE
    If (CandCnt>0)
      Y2 := ROVI_SOLVE()
      If (Y2[0]≟10000.)
        SubPrgResult := rovi_err
        Wait Sleep waitTime=999999
  UF := Y2
  Folder PICK_POS
    gGD_2_LM_p := pose_add(gGD_2_LM_RX, gGD_2_LM_Offset)
    gGD_2_M_p := pose_add(gGD_2_M_RX, gGD_2_M_Offset)
    gGD_2_RM_p := pose_add(gGD_2_RM_RX, gGD_2_RM_Offset)
  Folder CHECK_PICK_POS
    If (0≤DistPillar and DistPillar≤DistPillarAPTh)
      gGD_2_p := gGD_2_LM_p
    ElseIf (-DistPillarAPTh≤DistPillar and DistPillar≤0)
      gGD_2_p := gGD_2_RM_p
    Else 
      gGD_2_p := gGD_2_M_p
    PickPosFlange := GET_DEST_FLANGE(gGD_2_p, UF, PickTCP)
    PickPosDist := GET_DIST(PickPosFlange, p[0, 0, 0, 0, 0, 0])
    If ( not CHECK_DIST_NEAR(PickPosFlange, p[0, 0, 0, 0, 0, 0], RBArmLength+RBArmOffset))
      SubPrgResult := 923
      Wait Sleep waitTime=999999
  Folder PICK
    SetPayload (workpieceName=k10)
    BucketDef := pBucket[WorkPosNo]
    If (CaptIndexWk≟1)
      If ((BucketDef[2]+Sub104_TiltZTh[0]<CurrPos[2]) and (CurrPos[2]<BucketDef[2]+Sub104_TiltZTh[1]))
        If (0≤DistPillar and DistPillar≤DistPillarAPTh)
          SuppressedNode
            MoveL speed 200 mm/s, acceleration 70 mm/s^2 (useActiveTCP=false) tcp=TCP_1; feature=Bucket
              Waypoint TiltL (Relative): relativeFromPosition TCP in base x=-335.02 y=-289.975 z=399.986 mm, rx=-2.1962 ry=-2.2464 rz=-0.0001 rad; joints [-125.137, -72.094, -90.48, -107.417, 89.921, 53.694] deg; TCP offset x=0 y=80 z=420 mm, rx=0 ry=0 rz=0 rad; TCP in base x=-335.069 y=-289.996 z=400.008 mm, rx=2.1521 ry=2.2 rz=-0.0901 rad; joints [-128.746, -69.644, -93.066, -103.58, 93.161, 50.22] deg; feature pose in base x=326.04 y=491.74 z=0 mm, rx=0 ry=0 rz=-1.5932 rad
        Else 
          If WorkPosNo≟0
            MoveL speed 200 mm/s, acceleration 70 mm/s^2 (useActiveTCP=false) tcp=TCP_1; feature=Bucket
              Waypoint SlideL0 (Relative): relativeFromPosition TCP in base x=6.559 y=-389.302 z=60.921 mm, rx=-0.5073 ry=3.0586 rz=-0.014 rad; joints [-67.114, -66.849, -128.346, -73.737, 92.151, 4.181] deg; TCP in base x=6.579 y=-439.267 z=60.918 mm, rx=-0.5073 ry=3.0586 rz=-0.0139 rad; joints [-69.434, -72.805, -124.655, -71.563, 92.167, 1.857] deg
          Else 
            MoveL speed 200 mm/s, acceleration 70 mm/s^2 (useActiveTCP=false) tcp=TCP_1; feature=Bucket
              Waypoint SlideL1 (Relative): relativeFromPosition TCP in base x=-4.128 y=-329.518 z=106.532 mm, rx=-0.0229 ry=-3.1387 rz=-0.0019 rad; joints [-65.843, -58.986, -127.487, -83.647, 89.896, 25.103] deg; TCP in base x=-4.138 y=-279.531 z=106.538 mm, rx=-0.0228 ry=-3.1387 rz=-0.0019 rad; joints [-62.192, -52.298, -130.125, -87.703, 89.931, 28.744] deg
    ElseIf (CaptIndexWk≟2)
      If ((BucketDef[2]+Sub104_TiltZTh[0]<CurrPos[2]) and (CurrPos[2]<BucketDef[2]+Sub104_TiltZTh[1]))
        If (-DistPillarAPTh≤DistPillar and DistPillar≤0)
          SuppressedNode
            MoveL speed 200 mm/s, acceleration 70 mm/s^2 (useActiveTCP=false) tcp=TCP_1; feature=Bucket
              Waypoint TiltR (Relative): relativeFromPosition TCP in base x=-335.043 y=289.982 z=399.99 mm, rx=-2.1963 ry=-2.2462 rz=0.0001 rad; joints [-194.945, -71.897, -90.609, -107.481, 89.926, -16.106] deg; TCP in base x=-335.051 y=289.972 z=400.009 mm, rx=-2.152 ry=-2.1999 rz=-0.0898 rad; joints [-189.439, -69.266, -92.671, -107.022, 85.13, -10.62] deg
        Else 
          If WorkPosNo≟0
            MoveL speed 200 mm/s, acceleration 70 mm/s^2 (useActiveTCP=false) tcp=TCP_1; feature=Bucket
              Waypoint SlideR0 (Relative): relativeFromPosition TCP in base x=6.531 y=-439.223 z=60.88 mm, rx=-0.5073 ry=3.0587 rz=-0.0137 rad; joints [-69.436, -72.808, -124.656, -71.567, 92.166, 1.857] deg; TCP in base x=6.589 y=-389.288 z=60.942 mm, rx=-0.5074 ry=3.0586 rz=-0.014 rad; joints [-67.112, -66.85, -128.343, -73.741, 92.153, 4.181] deg
          Else 
            MoveL speed 200 mm/s, acceleration 70 mm/s^2 (useActiveTCP=false) tcp=TCP_1; feature=Bucket
              Waypoint SlideR1 (Relative): relativeFromPosition TCP in base x=-4.121 y=-279.485 z=106.522 mm, rx=-0.0229 ry=-3.1387 rz=-0.0021 rad; joints [-62.196, -52.302, -130.125, -87.705, 89.936, 28.743] deg; TCP in base x=-4.165 y=-329.432 z=106.437 mm, rx=-0.0229 ry=-3.1386 rz=-0.0022 rad; joints [-65.843, -58.989, -127.494, -83.649, 89.896, 25.103] deg
    If (0≤DistPillar and DistPillar≤DistPillarAPTh)
      SetPayload (workpieceName=k120)
      MoveL speed 400 mm/s, acceleration 70 mm/s^2 (useActiveTCP=false) tcp=TCP_RX; feature=UF
        Waypoint Variable (Variable): variable(featureName=gGD_4_LM)
      MoveL speed 250 mm/s, acceleration 50 mm/s^2 (useActiveTCP=false) tcp=TCP_RX; feature=UF
        Waypoint Variable (Variable): variable(featureName=gGD_3_LM_RX)
        SuppressedNode
          Waypoint Variable (Variable): variable(featureName=gGD_2_LM_RX)
        Waypoint Variable (Variable): variable=gGD_2_LM_p
        Set SingleDigitalPulseActionState SingleDigitalPulseActionState(hiPulseInSeconds=1, pin=GP_bool_out[14])
        Wait Sleep waitTime=0.5
        SetPayload (workpieceName=k10)
        SuppressedNode
          Popup Message (haltProgram=false message=ok? inputType=Text)
      Timer (action=Reset) variable(name=tm_handin)
      Timer (action=Start) variable=tm_handin
      Set DigitalOutput pin=digital_out[1]; digitalValue=1
      Force Frame feature=Joint_6_name; selection=[1, 1, 1, 0, 0, 0]; wrench=[0, 0, 20, 0, 0, 0]; limitsForce=[0.005, 0.005, 0.04, 0.034907, 0.034907, 1.047198]; limitsMotion=[0.1, 0.1, 0.1, 0.349066, 0.349066, 0.349066]
        SuppressedNode
          Wait Condition expression=((Currpos_p_UF0[1]≤(gGD_2_LM_RX[1]-HandInZ)) or (tm_handin>GPII_TMHandIn))
        Wait Condition expression=((Currpos_p_UF0[0]>(gGD_2_LM_p[0]+HandInZ)) or (tm_handin>GPII_TMHandIn))
      Timer (action=Stop) variable=tm_handin
      Set SingleDigitalPulseActionState SingleDigitalPulseActionState(hiPulseInSeconds=1, pin=GP_bool_out[15])
      Set DigitalOutput pin=digital_out[1]; digitalValue=0
    ElseIf (-DistPillarAPTh≤DistPillar and DistPillar≤0)
      SetPayload (workpieceName=k120)
      MoveL speed 400 mm/s, acceleration 70 mm/s^2 (useActiveTCP=false) tcp=TCP_RX; feature=UF
        Waypoint Variable (Variable): variable(featureName=gGD_4_RM)
      MoveL speed 250 mm/s, acceleration 50 mm/s^2 (useActiveTCP=false) tcp=TCP_RX; feature=UF
        Waypoint Variable (Variable): variable(featureName=gGD_3_RM_RX)
        SuppressedNode
          Waypoint Variable (Variable): variable(featureName=gGD_2_RM_RX)
        Waypoint Variable (Variable): variable=gGD_2_RM_p
        Set SingleDigitalPulseActionState SingleDigitalPulseActionState(hiPulseInSeconds=1, pin=GP_bool_out[14])
        Wait Sleep waitTime=0.5
        SetPayload (workpieceName=k10)
        SuppressedNode
          Popup Message (haltProgram=false message=ok? inputType=Text)
      Timer (action=Reset) variable=tm_handin
      Timer (action=Start) variable=tm_handin
      Set DigitalOutput pin=digital_out[1]; digitalValue=1
      Force Frame feature=Joint_6_name; selection=[1, 1, 1, 0, 0, 0]; wrench=[0, 0, 20, 0, 0, 0]; limitsForce=[0.005, 0.005, 0.04, 0.034907, 0.034907, 1.047198]; limitsMotion=[0.1, 0.1, 0.1, 0.349066, 0.349066, 0.349066]
        SuppressedNode
          Wait Condition expression=((Currpos_p_UF0[1]≤(gGD_2_RM_RX[1]-HandInZ)) or (tm_handin>GPII_TMHandIn))
        Wait Condition expression=((Currpos_p_UF0[0]>(gGD_2_RM_p[0]+HandInZ)) or (tm_handin>GPII_TMHandIn))
      Timer (action=Stop) variable=tm_handin
      Set SingleDigitalPulseActionState SingleDigitalPulseActionState(hiPulseInSeconds=1, pin=GP_bool_out[15])
      Set DigitalOutput pin=digital_out[1]; digitalValue=0
    Else 
      SetPayload (workpieceName=k120)
      MoveL speed 400 mm/s, acceleration 70 mm/s^2 (useActiveTCP=false) tcp=TCP_RX; feature=UF
        Waypoint Variable (Variable): variable(featureName=gGD_3_M_RX)
        SuppressedNode
          Waypoint Variable (Variable): variable(featureName=gGD_2_M_RX)
        Waypoint Variable (Variable): variable=gGD_2_M_p
        Set SingleDigitalPulseActionState SingleDigitalPulseActionState(hiPulseInSeconds=1, pin=GP_bool_out[14])
        Wait Sleep waitTime=0.5
        SetPayload (workpieceName=k10)
        SuppressedNode
          Popup Message (haltProgram=false message=ok? inputType=Text)
      Timer (action=Reset) variable=tm_handin
      Timer (action=Start) variable=tm_handin
      Set DigitalOutput pin=digital_out[1]; digitalValue=1
      Force Frame feature=Joint_6_name; selection=[1, 1, 1, 0, 0, 0]; wrench=[0, 0, 20, 0, 0, 0]; limitsForce=[0.005, 0.005, 0.04, 0.034907, 0.034907, 1.047198]; limitsMotion=[0.1, 0.1, 0.1, 0.349066, 0.349066, 0.349066]
        ShakeCnt := -1
        Loop While (checkContinuously=false) expression=((Currpos_p_UF0[0]≤(gGD_2_LM_p[0]+HandInZ)) and (tm_handin<GPII_TMHandIn))
          If UseShake
            If ShakeCnt<0
              Folder NOT_SHAKE
                Timer (action=Start) variable(name=tm_104)
                Wait Condition expression=tm_104>ShakeWaitSec
                Timer (action=Stop) variable=tm_104
                Timer (action=Reset) variable=tm_104
              ShakeCnt := 0
            IsShake := False
            Folder MONITOR_SPEED
              Timer (action=Reset) variable=tm_104
              If norm(TCPSpeed[1])<TCPSpeedThZ
                IsShake := True
                If ShakeCnt≟0
                  Timer (action=Start) variable=tm_104
                  Loop While (checkContinuously=false) expression=((tm_104<1.0) and (IsShake≟ True ))
                    If norm(TCPSpeed[1])≥TCPSpeedThZ
                      IsShake := False
                  Timer (action=Stop) variable=tm_104
                ShakeCnt := ShakeCnt+1
            Folder SHAKE
              If IsShake
                Sub3100_Option := 7
                Loop Counting (count=2) loopVariable(name=ループ_8)
                  '7:RX+,8:RX-,9:RY+,10:RY-,11:RZ+,12:RZ-'
                  Sub3100_Xd := [0.,0.,0.,0.,0.,0.]
                  Sub3100_q := floor((Sub3100_Option-1) / 2)
                  Sub3100_e := 1-((Sub3100_Option-1) % 2)*2
                  Sub3100_t := 0.2
                  Script: Sub3100_Xd[Sub3100_q]=d2r(Sub3100_XdRot/2.0)*Sub3100_e
                  Script: speedl(Sub3100_Xd,Sub3100_aRot/2.0,Sub3100_t)
                  If Sub3100_Option≟7
                    Sub3100_Option := 8
                  Else 
                    Sub3100_Option := 7
                  Wait Sleep waitTime=0.1
                IsShake := False
          Wait Sleep waitTime=0.1
      Set DigitalOutput pin=digital_out[1]; digitalValue=0
      Timer (action=Stop) variable=tm_handin
      Set SingleDigitalPulseActionState SingleDigitalPulseActionState(hiPulseInSeconds=1, pin=GP_bool_out[15])
      SuppressedNode
        IsSteady_01 := is_steady()
      SuppressedNode
        Wait Sleep waitTime=2
      SuppressedNode
        IsSteady_02 := is_steady()
    Timer (action=Reset) variable(name=tm_steady_104)
    Timer (action=Start) variable=tm_steady_104
    Wait Condition expression=is_steady()
    Timer (action=Stop) variable=tm_steady_104
    SuppressedNode
      Popup Message (haltProgram=false message=force done! inputType=Text)
    If ( not GPBI_WorkExists)
      SetPayload (workpieceName=k10)
      If (0≤DistPillar and DistPillar≤DistPillarAPTh)
        MoveL speed 400 mm/s, acceleration 140 mm/s^2 (useActiveTCP=false) tcp=TCP_RX; feature=UF
          SuppressedNode
            Waypoint Variable (Variable): variable(featureName=gGD_2_LM_RX)
          Waypoint Variable (Variable): variable=gGD_2_LM_p
          Waypoint Variable (Variable): variable(featureName=gGD_3_LM_RX)
        MoveL speed 400 mm/s, acceleration 140 mm/s^2 (useActiveTCP=false) tcp=TCP_RX; feature=UF
          Waypoint Variable (Variable): variable(featureName=gGD_4_LM)
      ElseIf (-DistPillarAPTh≤DistPillar and DistPillar≤0)
        MoveL speed 400 mm/s, acceleration 70 mm/s^2 (useActiveTCP=false) tcp=TCP_RX; feature=UF
          SuppressedNode
            Waypoint Variable (Variable): variable(featureName=gGD_2_RM_RX)
          Waypoint Variable (Variable): variable=gGD_2_RM_p
          Waypoint Variable (Variable): variable(featureName=gGD_3_RM_RX)
        MoveL speed 400 mm/s, acceleration 70 mm/s^2 (useActiveTCP=false) tcp=TCP_RX; feature=UF
          Waypoint Variable (Variable): variable(featureName=gGD_4_RM)
      Else 
        MoveL speed 400 mm/s, acceleration 70 mm/s^2 (useActiveTCP=false) tcp=TCP_RX; feature=UF
          SuppressedNode
            Waypoint Variable (Variable): variable(featureName=gGD_2_M_RX)
          Waypoint Variable (Variable): variable=gGD_2_M_p
          Waypoint Variable (Variable): variable(featureName=gGD_3_M_RX)
      SetPayload (workpieceName=k25)
      Folder ROVI_CAPTURE
        CaptPos := GET_CAPTPOS()
        MoveJ speed 40 deg/s, acceleration 20 deg/s^2 (useActiveTCP=false) tcp=TCP_1; feature=Bucket
          Waypoint Variable (Variable): variable=CaptPos
        Folder BUCKET
          Script: SET_BUCKET_DEF()
          BucketUpperPos := GET_BUCKET_UPPER()
        MoveJ speed 40 deg/s, acceleration 20 deg/s^2 (useActiveTCP=false) tcp=TCP_1; feature=Bucket
          Waypoint Variable (Variable): variable=BucketUpperPos
        Wait Sleep waitTime=1
        SuppressedNode
          Script: POPUP_CAPT_OPTION()
      SubPrgResult := 821
      Wait Sleep waitTime=999999
SubProgram SUB_105 (keepSynchronizedWithDisk=true) programFile=/programs/GD/SUB_105.urp
  UF := Y2
  Folder PICK
    Folder FREE_DRIVE
      SetPayload (workpieceName=k2)
      Script: freedrive_mode()
      Set NoAction tcp=ZERO
      Wait Sleep waitTime=0.5
      Script: end_freedrive_mode()
    Script: force_mode_set_gain_scaling(0.9)
    Set SingleDigitalPulseActionState SingleDigitalPulseActionState(hiPulseInSeconds=1, pin=GP_bool_out[15])
    ForceStartZ := CurrPos_p[2]
    If LevelZ<0
      CutOffZ := 0.0
    Else 
      CutOffZ := LevelZ
    CutOffZAdd := NeighborZ+BeyondZ
    SuppressedNode
      Popup Message (haltProgram=false message=zero ft_sensor... inputType=Text)
    TCPForceBak := TCPForce
    Timer (action=Reset) variable(name=tm_cutoff)
    Timer (action=Start) variable=tm_cutoff
    SuppressedNode
      If (0≤DistPillar and DistPillar≤DistPillarCOTh) removedSiblings(If(type=ElseIf checkContinuously=false, expression=(-DistPillarCOTh≤DistPillar and DistPillar≤0), children(Set(type=DigitalOutput, pin=digital_out[2], digitalValue=1), SuppressedNode(suppressedNode(type=Frame, feature=Bucket, selection=[1, 1, 1, 1, 1, 1], wrench=[-40, 0, 40, 0, 0, 0], limitsForce=[0.01, 0.01, 0.015, 0.174533, 0.174533, 0.174533], limitsMotion=[0.1, 0.1, 0.1, 0.349066, 0.349066, 0.349066], children(SetPayload(workpieceName=k05), Assignment(valueSource=Expression, variable=CutOffZ, expression=CutOffZ+CutOffZAdd), Wait(type=Condition, expression=tm_cutoff>GPII_TMCutOff or CurrPos_p[2]>ForceStartZ+CutOffZ or GPBI_BLLoad2)))), Folder(name=FORCE_CUTOFF, children(SetPayload(workpieceName=k1), Wait(type=Sleep, waitTime=0.02), SuppressedNode(suppressedNode(type=Line, expression=zero_ftsensor())), Assignment(valueSource=Expression, variable=ForceFeature, expression=Bucket), Assignment(valueSource=Expression, variable=ForceValue, expression=[-40,0,40,0,0,0]), Assignment(valueSource=Expression, variable=ForceLimit, expression=[0.01,0.01,ForceLimitZ[0],d2r(10.),d2r(10.),d2r(10.)]), Assignment(valueSource=Expression, variable=CutOffZ, expression=CutOffZ+CutOffZAdd), Script(type=Line, expression=force_mode(ForceFeature,ForceAxis,ForceValue,ForceType,ForceLimit)), Loop(type=While checkContinuously=true, expression=tm_cutoff<GPII_TMCutOff and CurrPos_p[2]<ForceStartZ+CutOffZ and ( not GP_bool_in[11]), children(If(type=If checkContinuously=false, expression=UseRZSuppress, children(If(type=If checkContinuously=false, expression=WorkPosNo≟0, children(Script(type=Line, expression=ForceValue[5]=-GET_FORCE_VALUE_RZ(g2GD_pos5)))), If(type=ElseIf checkContinuously=false, expression=WorkPosNo≟1, children(Script(type=Line, expression=ForceValue[5]=-GET_FORCE_VALUE_RZ(g1GD_pos5)))), Script(type=Line, expression=force_mode(ForceFeature,ForceAxis,ForceValue,ForceType,ForceLimit)))), Script(type=Line, expression=sync()))), Script(type=Line, expression=end_force_mode()), Script(type=Line, expression=stopl(1.0)))), Set(type=DigitalOutput, pin=digital_out[3], digitalValue=0))), SuppressedNode(suppressedNode(type=Else checkContinuously=false, children(Set(type=DigitalOutput, pin=digital_out[3], digitalValue=1), SuppressedNode(suppressedNode(type=Frame, feature=Bucket, selection=[1, 1, 1, 1, 1, 1], wrench=[0, 0, 40, 0, 0, 0], limitsForce=[0.01, 0.01, 0.015, 0.174533, 0.174533, 0.174533], limitsMotion=[0.1, 0.1, 0.1, 0.349066, 0.349066, 0.349066], children(SetPayload(workpieceName=k05), SuppressedNode(suppressedNode(valueSource=Expression, variable=CutOffZ, expression=CutOffZ+CutOffZDef)), Assignment(valueSource=Expression, variable=CutOffZ, expression=CutOffZ+CutOffZAdd), Wait(type=Condition, expression=tm_cutoff>GPII_TMCutOff or CurrPos_p[2]>ForceStartZ+CutOffZ or GPBI_BLLoad2)))), Folder(name=FORCE_CUTOFF, children(SetPayload(workpieceName=k1), Wait(type=Sleep, waitTime=0.02), SuppressedNode(suppressedNode(type=Line, expression=zero_ftsensor())), Assignment(valueSource=Expression, variable=ForceStep, expression=0), Assignment(valueSource=Expression, variable=ForceValue, expression=[0,0,40,0,0,0]), Assignment(valueSource=Expression, variable=ForceFeature, expression=Bucket), Assignment(valueSource=Expression, variable=CutOffZ, expression=CutOffZ+CutOffZAdd), Loop(type=While checkContinuously=false, expression=tm_cutoff<GPII_TMCutOff, children(If(type=If checkContinuously=false, expression=WorkPosNo≟0, children(Script(type=Line, expression=ForceValue[5]=-GET_FORCE_VALUE_RZ(g2GD_pos5)))), If(type=ElseIf checkContinuously=false, expression=WorkPosNo≟1, children(Script(type=Line, expression=ForceValue[5]=-GET_FORCE_VALUE_RZ(g1GD_pos5)))), Switch(expression=ForceStep, children(Case(caseValue=0, children(Assignment(valueSource=Expression, variable=ForceStep, expression=1), Assignment(valueSource=Expression, variable=ForceLimit, expression=[0.01,0.01,ForceLimitZ[ForceStep-1],d2r(10.),d2r(10.),d2r(10.)]), Script(type=Line, expression=force_mode(ForceFeature,ForceAxis,ForceValue,ForceType,ForceLimit)))), Case(caseValue=1, children(If(type=If checkContinuously=false, expression=GPBI_BLLoad1, children(Assignment(valueSource=Expression, variable=ForceStep, expression=2), Assignment(valueSource=Expression, variable=ForceLimit, expression=[0.01,0.01,ForceLimitZ[ForceStep-1],d2r(10.),d2r(10.),d2r(10.)]), Script(type=Line, expression=force_mode(ForceFeature,ForceAxis,ForceValue,ForceType,ForceLimit)))), If(type=ElseIf checkContinuously=false, expression=UseRZSuppress, children(Script(type=Line, expression=force_mode(ForceFeature,ForceAxis,ForceValue,ForceType,ForceLimit)))))), Case(caseValue=2, children(If(type=If checkContinuously=false, expression=GP_bool_in[11], children(Script(type=Line, expression=break))), If(type=If checkContinuously=false, expression=CurrPos_p[2]>ForceStartZ+CutOffZ, children(Assignment(valueSource=Expression, variable=ForceStep, expression=3), Script(type=Line, expression=ForceValue[2]=0.0), Assignment(valueSource=Expression, variable=ForceLimit, expression=[0.01,0.01,ForceLimitZ[ForceStep-1],d2r(10.),d2r(10.),d2r(10.)]), Script(type=Line, expression=force_mode(ForceFeature,ForceAxis,ForceValue,ForceType,ForceLimit)))), If(type=ElseIf checkContinuously=false, expression=UseRZSuppress, children(Script(type=Line, expression=force_mode(ForceFeature,ForceAxis,ForceValue,ForceType,ForceLimit)))))), Case(caseValue=3, children(If(type=If checkContinuously=false, expression=GP_bool_in[11], children(Script(type=Line, expression=break))), If(type=If checkContinuously=false, expression=(UseRZSuppress and (ForceValue[5]≠0.0)), children(Script(type=Line, expression=force_mode(ForceFeature,ForceAxis,ForceValue,ForceType,ForceLimit)))), If(type=Else checkContinuously=false, children(If(type=If checkContinuously=false, expression=CHECK_SPEED(StopSpeed) and ((UseRZSuppress and (ForceValue[5]==0.0)) or ( not UseRZSuppress)), children(Script(type=Line, expression=break))))))), SuppressedNode(suppressedNode(caseValue=4, children(Assignment(valueSource=Expression, variable(name=var_9), expression=var_9+1), If(type=If checkContinuously=false, expression=CHECK_SPEED(StopSpeed), children(Script(type=Line, expression=break)))))))), Script(type=Line, expression=sync()))), Script(type=Line, expression=end_force_mode()), Script(type=Line, expression=stopl(5.0)))), Set(type=DigitalOutput, pin=digital_out[3], digitalValue=0)))))
        Set DigitalOutput pin=digital_out[3]; digitalValue=1
        SuppressedNode
          Force Frame feature=Bucket; selection=[1, 1, 1, 1, 1, 1]; wrench=[40, 0, 40, 0, 0, 0]; limitsForce=[0.01, 0.01, 0.015, 0.174533, 0.174533, 0.174533]; limitsMotion=[0.1, 0.1, 0.1, 0.349066, 0.349066, 0.349066]
            SetPayload (workpieceName=k05)
            CutOffZ := CutOffZ+CutOffZAdd
            Wait Condition expression=tm_cutoff>GPII_TMCutOff or CurrPos_p[2]>ForceStartZ+CutOffZ or GPBI_BLLoad2
        Folder FORCE_CUTOFF
          SetPayload (workpieceName=k1)
          Wait Sleep waitTime=0.02
          SuppressedNode
            Script: zero_ftsensor()
          ForceFeature := Bucket
          ForceValue := [40,0,40,0,0,0]
          ForceLimit := [0.01,0.01,ForceLimitZ[0],d2r(10.),d2r(10.),d2r(10.)]
          CutOffZ := CutOffZ+CutOffZAdd
          Script: force_mode(ForceFeature,ForceAxis,ForceValue,ForceType,ForceLimit)
          Loop While (checkContinuously=true) expression=tm_cutoff<GPII_TMCutOff and CurrPos_p[2]<ForceStartZ+CutOffZ and ( not GP_bool_in[11])
            If UseRZSuppress
              If WorkPosNo≟0
                Script: ForceValue[5]=-GET_FORCE_VALUE_RZ(g2GD_pos5)
              ElseIf WorkPosNo≟1
                Script: ForceValue[5]=-GET_FORCE_VALUE_RZ(g1GD_pos5)
              Script: force_mode(ForceFeature,ForceAxis,ForceValue,ForceType,ForceLimit)
            Script: sync()
          Script: end_force_mode()
          Script: stopl(1.0)
        Set DigitalOutput pin=digital_out[3]; digitalValue=0
    Set DigitalOutput pin=digital_out[3]; digitalValue=1
    Folder FORCE_CUTOFF
      SetPayload (workpieceName=kjF)
      Wait Sleep waitTime=0.02
      SuppressedNode
        Script: zero_ftsensor()
      ForceStep := 0
      If (0≤DistPillar and DistPillar≤DistPillarCOTh)
        ForceValue := [40,0,60,0,0,0]
      ElseIf (-DistPillarCOTh≤DistPillar and DistPillar≤0)
        ForceValue := [-40,0,60,0,0,0]
      Else 
        ForceValue := [0,0,60,0,0,0]
      ForceFeature := Bucket
      ForceLZDecayWk := 0
      ForceVZDecayWk := 0
      CutOffZ := CutOffZ+CutOffZAdd
      Timer (action=Reset) variable(name=tm_decay)
      Loop While (checkContinuously=false) expression=tm_cutoff<GPII_TMCutOff
        If WorkPosNo≟0
          Script: ForceValue[5]=-GET_FORCE_VALUE_RZ(g2GD_pos5)
        ElseIf WorkPosNo≟1
          Script: ForceValue[5]=-GET_FORCE_VALUE_RZ(g1GD_pos5)
        Switch expression=ForceStep
          Case (caseValue=0)
            ForceStep := 1
            ForceLimit := [0.01,0.01,ForceLimitZ[ForceStep-1],d2r(10.),d2r(10.),d2r(10.)]
            Script: force_mode(ForceFeature,ForceAxis,ForceValue,ForceType,ForceLimit)
          Case (caseValue=1)
            If GPBI_BLLoad1
              ForceStep := 2
              ForceLimit := [0.01,0.01,ForceLimitZ[ForceStep-1],d2r(10.),d2r(10.),d2r(10.)]
              Script: force_mode(ForceFeature,ForceAxis,ForceValue,ForceType,ForceLimit)
            ElseIf UseRZSuppress
              Script: force_mode(ForceFeature,ForceAxis,ForceValue,ForceType,ForceLimit)
          Case (caseValue=2)
            If GPBI_BLLoad2
              Script: break
            Script: ForceValue[2]=ForceValue[2]-ForceVZDecayWk
            Script: ForceLimit[2]=ForceLimit[2]-ForceLZDecayWk
            If (ForceValue[2]≤0 and ForceLZDecay≟0)
              Timer (action=Stop) variable=tm_decay
              ForceStep := 3
              Script: break
            ElseIf (ForceLimit[2]≤StopSpeed[2] and ForceVZDecay≟0)
              Timer (action=Stop) variable=tm_decay
              ForceStep := 3
              Script: break
            ElseIf (ForceValue[2]≤0 and ForceLimit[2]≤0)
              Timer (action=Stop) variable=tm_decay
              ForceStep := 3
              Script: break
            ElseIf (( CurrPos_p[2]>ForceStartZ+CutOffZ ) or ( not CHECK_DIST_NEAR(CurrPos, p[0,0,0,0,0,0], RBArmLength)))
              Timer (action=Start) variable=tm_decay
              TCPForceBak2 := TCPForce
              TCPSpeedBak2 := TCPSpeed
              Script: ForceValue[0]=0.0
              If (ForceVZDecay≟0 and ForceLZDecay≟0)
                ForceVZDecayWk := ForceValue[2]
                ForceLZDecayWk := 0
              ElseIf (ForceVZDecay≠0 and ForceLZDecay≟0)
                ForceVZDecayWk := ForceVZDecay
                ForceLZDecayWk := 0
              ElseIf (ForceVZDecay≟0 and ForceLZDecay≠0)
                ForceVZDecayWk := 0
                ForceLZDecayWk := ForceLZDecay
              Else 
                ForceVZDecayWk := ForceVZDecay
                ForceLZDecayWk := ForceLZDecay
              Script: force_mode(ForceFeature,ForceAxis,ForceValue,ForceType,ForceLimit)
            ElseIf UseRZSuppress
              If (ForceValue[2]<0)
                Script: ForceValue[2]=0.0
              If (ForceLimit[2]≤StopSpeed[2])
                Script: ForceLimit[2]=StopSpeed[2]
              Script: force_mode(ForceFeature,ForceAxis,ForceValue,ForceType,ForceLimit)
          Case (caseValue=3)
            If GPBI_BLLoad2
              Script: break
            If (UseRZSuppress and (ForceValue[5]≠0.0))
              Script: force_mode(ForceFeature,ForceAxis,ForceValue,ForceType,ForceLimit)
            Else 
              If CHECK_SPEED(StopSpeed) and ((UseRZSuppress and (ForceValue[5]==0.0)) or ( not UseRZSuppress))
                Script: break
          SuppressedNode
            Case (caseValue=4)
              var_9 := var_9+1
              If CHECK_SPEED(StopSpeed)
                Script: break
        Script: sync()
      Script: end_force_mode()
      Script: stopl(5.0)
    SuppressedNode
      Wait NoWait
    SuppressedNode
      Script: end_force_mode()
    SuppressedNode
      Script: stopl(1.0)
    Set DigitalOutput pin=digital_out[3]; digitalValue=0
    SuppressedNode
      Wait Condition expression=is_steady()
    Timer (action=Stop) variable=tm_cutoff
  If (GPBI_BLLoad2)
    SubPrgResult := 825
    Wait Sleep waitTime=999999
  If ( not GPBI_BLLoad1)
    SubPrgResult := 822
    Wait Sleep waitTime=999999
  SetPayload (workpieceName=k10)
  SuppressedNode
    IsSteady_01 := is_steady()
  SuppressedNode
    Wait Sleep waitTime=1
  SuppressedNode
    IsSteady_02 := is_steady()
  Timer (action=Reset) variable(name=tm_steady_105)
  Timer (action=Start) variable=tm_steady_105
  SuppressedNode
    Wait Condition expression=is_steady()
  Timer (action=Stop) variable=tm_steady_105
  Set DigitalOutput pin=digital_out[0]; digitalValue=1
  Folder FREE_DRIVE
    Script: freedrive_mode()
    SetPayload (workpieceName=k2)
    Set NoAction tcp=ZERO
    Wait Sleep waitTime=1.5
    Script: end_freedrive_mode()
  Wait Condition expression=is_steady()
  Set DigitalOutput pin=digital_out[0]; digitalValue=0
  Folder CHK_RX_TILT
    If UseChkRXTilt
      Set NoAction tcp=TCP_1
      Script: sync()
      Script: CurrPos_p=get_actual_tcp_pose()
      CurrposAligned := p[0,0,0,0,0,0]
      CurrposAligned := GET_ALIGNED_TCP(CurrposAligned)
      If (not CHECK_RX_TILT(CurrposAligned))
        SubPrgResult := 825
        Wait Sleep waitTime=999999
  Folder CV_CORR_RZ
    If UseCVCorr
      Set NoAction tcp=TCP_1
      Script: sync()
      Script: CurrPos_p=get_actual_tcp_pose()
      CurrposAligned := p[0,0,0,0,0,0]
      CurrposAligned := GET_ALIGNED_TCP(CurrposAligned)
      Script: GET_CVCORR_VALUE(CurrposAligned)
  Folder CUTOFF_POSE
    If UseCutOffTCP
      Set NoAction tcp=TCP_1
      CutOffPos := p[0.,0.,0.,0.,0.,0.]
      CutOffPos := GET_ALIGNED_TCP(CutOffPos)
      CutOffTCP := pose_trans(pose_inv(CurrPos),CutOffPos)
      Set NoAction tcp=ZERO
      CutOffTCP := pose_trans(get_tcp_offset(),CutOffTCP)
      Set NoAction tcp=TCP_1
    Else 
      Set NoAction tcp=TCP_1
      CutOffTCP := get_tcp_offset()
SubProgram SUB_106 (keepSynchronizedWithDisk=true) programFile=/programs/GD/SUB_106.urp
  If GPBI_WorkExists (checkContinuously=true)
    Folder TRANSFER
      Set DigitalOutput pin=digital_out[7]; digitalValue=1
      SetPayload (workpieceName=k120)
      If UseZRotate
        Set NoAction tcp=TCP_COG
        Script: sync()
        If UseBaseZRotate
          If (WorkPosNo≟0)
            gGD_pos5 := g2GD_pos5_NEAR
          ElseIf (WorkPosNo≟1)
            gGD_pos5 := g1GD_pos5_NEAR
          Script: CurrPos_p=get_actual_tcp_pose()
          MoveL speed 60 mm/s, acceleration 10 mm/s^2 (useActiveTCP=false) tcp=TCP_COG; feature=Base
            SuppressedNode
              PoseSub := pose_sub(CurrPos_p,g2GD_pos5_NEAR)
            PoseSub := pose_sub(CurrPos_p,gGD_pos5)
            RZSub := r2d(PoseSub[5])
            If (norm(PoseSub[5])≥d2r(RZTh))
              PoseAdd := pose_add(p[0,0,0,0,0,d2r(RZSub)],p[0,0,0,CurrPos_p[3],CurrPos_p[4],CurrPos_p[5]])
              PoseAdd := p[CurrPos_p[0],CurrPos_p[1],CurrPos_p[2],PoseAdd[3],PoseAdd[4],PoseAdd[5]]
              Waypoint Variable (Variable): variable=PoseAdd
        Else 
          If (WorkPosNo≟0)
            gGD_pos5 := g2GD_pos5
          ElseIf (WorkPosNo≟1)
            gGD_pos5 := g1GD_pos5
          MoveL speed 60 mm/s, acceleration 10 mm/s^2 (useActiveTCP=false) tcp=ZERO; feature=Base
            SuppressedNode
              PoseSub := pose_sub(CurrPos, pose_trans(g2GD_pos5, pose_inv(get_tcp_offset())))
            PoseSub := pose_sub(CurrPos, pose_trans(gGD_pos5, pose_inv(get_tcp_offset())))
            RZSub := r2d(PoseSub[5])
            If (norm(PoseSub[5])≥d2r(RZTh))
              Script: PoseSub[0]=0.0
              Script: PoseSub[1]=0.0
              Script: PoseSub[2]=0.0
              PoseAdd := pose_add(PoseSub, CurrPos)
              Waypoint Variable (Variable): variable=PoseAdd
      If UseCVCorr and UseCVCorrCam
        WorkNoOffset := WorkNoCV
        thrd108 := RUN_THREAD_ROVI()
      If (WorkPosNo≟0)
        SuppressedNode
          MoveL speed 250 mm/s, acceleration 50 mm/s^2 (useActiveTCP=false) tcp=TCP_1; feature=Base
            Waypoint Variable (Variable): variable(featureName=g2GD_pos5)
        Script: set_tcp(CutOffTCP)
        Script: sync()
        MoveL speed 250 mm/s, acceleration 25 mm/s^2 (useActiveTCP=true) feature=Base
          If UseZSlide
            gGD_pos5 := GET_ZSLIDE_POS(g2GD_pos5_NEAR)
          Else 
            gGD_pos5 := g2GD_pos5
          Script: DistBKUpper=GET_DIST(CurrPos_p,gGD_pos5)
          If ( not CHECK_DIST_NEAR(CurrPos_p, gGD_pos5, DistBKUpperTh))
            Waypoint Variable (Variable): variable=gGD_pos5
          Set DigitalOutput pin=digital_out[7]; digitalValue=0
        Set DigitalOutput pin=digital_out[6]; digitalValue=1
        MoveL speed 250 mm/s, acceleration 50 mm/s^2 (useActiveTCP=true) feature=Base
          SetPayload (workpieceName=k10)
          SuppressedNode
            Waypoint Variable (Variable): variable(featureName=g2GD_pos4)
          Waypoint Variable (Variable): motionParameters(blendRadius=0.1); variable(featureName=g2GD_pos3)
          SuppressedNode
            Waypoint Variable (Variable): motionParameters(jointSpeed=1.047198 jointAcceleration=1.396263 cartesianSpeed=0.4 cartesianAcceleration=0.07); variable(featureName=g2GD_pos2)
          PoseAdd := GET_CVCORR_POS(g2GD_pos2)
          Waypoint Variable (Variable): motionParameters(jointSpeed=1.047198 jointAcceleration=1.396263 cartesianSpeed=0.4 cartesianAcceleration=0.07); variable=PoseAdd
        Set DigitalOutput pin=digital_out[6]; digitalValue=0
        SuppressedNode
          Set DigitalOutput pin=digital_out[4]; digitalValue=1
        SuppressedNode
          MoveL speed 400 mm/s, acceleration 70 mm/s^2 (useActiveTCP=true) feature=Base
            SetPayload (workpieceName=k120)
            SuppressedNode
              Waypoint Variable (Variable): motionParameters(blendRadius=0.05); variable(featureName=g2GD_pos1)
            PoseAdd := GET_CVCORR_POS(g2GD_pos1)
            Waypoint Variable (Variable): motionParameters(blendRadius=0.05); variable=PoseAdd
      ElseIf (WorkPosNo≟1)
        SuppressedNode
          CircleMove (OrientationMode=UNCONSTRAINED)
        SuppressedNode
          Set NoAction tcp=TCP_COG
        SuppressedNode
          If UseBaseZRotate removedSiblings(If(type=Else checkContinuously=false, children(Move(motionType=MoveL speed=0.06 acceleration=0.01 useActiveTCP=false positionType=CartesianPose, tcp=ZERO, feature=Base, children(Assignment(valueSource=Expression, variable=PoseSub, expression=pose_sub(CurrPos, pose_trans(g1GD_pos5, pose_inv(get_tcp_offset())))), Assignment(valueSource=Expression, variable=RZSub, expression=r2d(PoseSub[5])), If(type=If checkContinuously=false, expression=(norm(PoseSub[5])≥d2r(RZTh)), children(Script(type=Line, expression=PoseSub[0]=0.0), Script(type=Line, expression=PoseSub[1]=0.0), Script(type=Line, expression=PoseSub[2]=0.0), Assignment(valueSource=Expression, variable=PoseAdd, expression=pose_add(PoseSub, CurrPos)), Waypoint(type=Variable name=Variable, variable=PoseAdd))))))))
            Script: sync()
            Script: CurrPos_p=get_actual_tcp_pose()
            MoveL speed 60 mm/s, acceleration 10 mm/s^2 (useActiveTCP=false) tcp=TCP_COG; feature=Base
              PoseSub := pose_sub(CurrPos_p,g1GD_pos5_NEAR)
              RZSub := r2d(PoseSub[5])
              If (norm(PoseSub[5])≥d2r(RZTh))
                PoseAdd := pose_add(p[0,0,0,0,0,d2r(RZSub)],p[0,0,0,CurrPos_p[3],CurrPos_p[4],CurrPos_p[5]])
                PoseAdd := p[CurrPos_p[0],CurrPos_p[1],CurrPos_p[2],PoseAdd[3],PoseAdd[4],PoseAdd[5]]
                Waypoint Variable (Variable): variable=PoseAdd
        SuppressedNode
          MoveL speed 250 mm/s, acceleration 50 mm/s^2 (useActiveTCP=false) tcp=TCP_1; feature=Base
            Waypoint Variable (Variable): variable(featureName=g1GD_pos5)
        Script: set_tcp(CutOffTCP)
        Script: sync()
        MoveL speed 250 mm/s, acceleration 38 mm/s^2 (useActiveTCP=true) feature=Base
          If UseZSlide
            gGD_pos5 := GET_ZSLIDE_POS(g1GD_pos5_NEAR)
          Else 
            gGD_pos5 := g1GD_pos5
          Script: DistBKUpper=GET_DIST(CurrPos_p,gGD_pos5)
          If ( not CHECK_DIST_NEAR(CurrPos_p, gGD_pos5, DistBKUpperTh))
            Waypoint Variable (Variable): variable=gGD_pos5
        Set DigitalOutput pin=digital_out[4]; digitalValue=0
        Set DigitalOutput pin=digital_out[6]; digitalValue=1
        MoveL speed 250 mm/s, acceleration 50 mm/s^2 (useActiveTCP=true) feature=Base
          SetPayload (workpieceName=k10)
          Waypoint Variable (Variable): variable(featureName=g1GD_pos4)
          Waypoint Variable (Variable): variable(featureName=g1GD_pos3)
          SuppressedNode
            Waypoint Variable (Variable): variable(featureName=g1GD_pos2)
          PoseAdd := GET_CVCORR_POS(g1GD_pos2)
          Waypoint Variable (Variable): variable=PoseAdd
        Set DigitalOutput pin=digital_out[6]; digitalValue=0
        SuppressedNode
          Set DigitalOutput pin=digital_out[4]; digitalValue=1
        SuppressedNode
          MoveL speed 400 mm/s, acceleration 140 mm/s^2 (useActiveTCP=true) feature=Base
            SetPayload (workpieceName=k120)
            SuppressedNode
              Waypoint Variable (Variable): motionParameters(blendRadius=0.1); variable(featureName=g1GD_pos1)
            PoseAdd := GET_CVCORR_POS(g1GD_pos1)
            Waypoint Variable (Variable): motionParameters(blendRadius=0.1); variable=PoseAdd
  SuppressedNode
    Set DigitalOutput pin=digital_out[4]; digitalValue=0
  If ( not GPBI_WorkExists)
    SubPrgResult := 820
    Wait Sleep waitTime=999999
SubProgram SUB_108 (keepSynchronizedWithDisk=true) programFile=/programs/GD/SUB_108.urp
  If UseCVCorr and UseCVCorrCam
    Script: JOIN_THREAD_ROVI(thrd108)
    If THREAD_ROVI_ERR≠0
      Folder ROVI_RECIPE
        If (not ROVI_RECIPE(GPII_WorkNo+WorkNoCV))
          SubPrgResult := rovi_err
          Wait Sleep waitTime=999999
      Folder ROVI_RESET
        If (not ROVI_RESET())
          SubPrgResult := rovi_err
          Wait Sleep waitTime=999999
      Folder ROVI_CAPTURE
        If ( not ROVI_CAPTURE())
          SubPrgResult := rovi_err
          Wait Sleep waitTime=999999
      Folder ROVI_SOLVE
        Y2 := ROVI_SOLVE()
        If (Y2[0]≟10000.)
          SubPrgResult := 824
          Wait Sleep waitTime=999999
    CutOffTCP := pose_trans(Y2, get_tcp_offset())
SubProgram SUB_121 (keepSynchronizedWithDisk=true) programFile=/programs/GD/SUB_121.urp
  Script: SET_CV()
  If GPBI_WorkExists (checkContinuously=true)
    SetPayload (workpieceName=k120)
    Script: set_tcp(CutOffTCP)
    Script: sync()
    MoveL speed 250 mm/s, acceleration 30 mm/s^2 (useActiveTCP=true) feature=CV
      SuppressedNode
        Waypoint Variable (Variable): variable(featureName=gCV_2_M)
      PoseAdd := GET_CVCORR_POS(gCV_2_M)
      Waypoint Variable (Variable): variable=PoseAdd
    SuppressedNode
      If GPBI_AllowGoCV≠ True
        SubPrgResult := 823
        Wait Sleep waitTime=999999
    Wait DigitalInput pin=GPBI_AllowGoCV; digitalValue=1
    Popup Message (haltProgram=false message=stop inputType=Text)
    MoveL speed 300 mm/s, acceleration 70 mm/s^2 (useActiveTCP=true) feature=CV
      SuppressedNode
        Waypoint Variable (Variable): variable(featureName=gCV_1_M)
      PoseAdd := GET_CVCORR_POS(gCV_1_M)
      Waypoint Variable (Variable): variable=PoseAdd
    Set NoAction tcp=TCP_1
    Popup Message (haltProgram=false message=stop inputType=Text)
    SuppressedNode
      Folder CV_CORR_RZ
        If UseCVCorr
          RZSub := CVCorrRZVal
          Set NoAction tcp=TCP_1
          Wait Sleep waitTime=0.02
          Script: CurrPos_p=get_actual_tcp_pose()
          MoveL speed 60 mm/s, acceleration 10 mm/s^2 (useActiveTCP=false) tcp=TCP_1; feature=Base
            PoseAdd := pose_add(p[0,0,0,0,0,d2r(-RZSub)],p[0,0,0,CurrPos_p[3],CurrPos_p[4],CurrPos_p[5]])
            PoseAdd := p[CurrPos_p[0],CurrPos_p[1],CurrPos_p[2],PoseAdd[3],PoseAdd[4],PoseAdd[5]]
            Waypoint Variable (Variable): variable=PoseAdd
  Set NoAction tcp=TCP_1
  If ( not GPBI_WorkExists)
    Script: stopl(1.2)
    SubPrgResult := 820
    Wait Sleep waitTime=999999
SubProgram SUB_122 (keepSynchronizedWithDisk=true) programFile=/programs/GD/SUB_122.urp
  Script: SET_CV()
  Set SingleDigitalPulseActionState SingleDigitalPulseActionState(hiPulseInSeconds=1, pin=GP_bool_out[15])
  SetPayload (workpieceName=k05)
  ForceStartZ := CurrPos[2]
  Timer (action=Reset) variable(name=tm_landed)
  Timer (action=Start) variable=tm_landed
  Set DigitalOutput pin=digital_out[5]; digitalValue=1
  Force Frame feature=CV; selection=[1, 1, 1, 0, 1, 0]; wrench=[0, 0, -40, 0, 0, 0]; limitsForce=[0.005, 0.005, 0.02, 0.174533, 0.034907, 0.174533]; limitsMotion=[0.1, 0.1, 0.1, 0.349066, 0.349066, 0.349066]
    Wait Condition expression=GPII_TMLanded<tm_landed or GPBI_BLLoad0 or CurrPos[2]<ForceStartZ-UnloadZ
    Wait Sleep waitTime=0.5
  Set DigitalOutput pin=digital_out[5]; digitalValue=0
  Script: end_force_mode()
  Timer (action=Stop) variable=tm_landed
  If ( not GPBI_BLLoad0)
    SubPrgResult := 824
    Wait Sleep waitTime=999999
  SetPayload (workpieceName=k10)
  MoveL speed 200 mm/s, acceleration 70 mm/s^2 (useActiveTCP=false) tcp=TCP_1; feature=CV
    Wait Sleep waitTime=1
    Waypoint Variable (Variable): motionParameters(jointSpeed=1.047198 jointAcceleration=1.396263 cartesianSpeed=0.03 cartesianAcceleration=0.03); variable(featureName=gCV_11_M)
    Waypoint Variable (Variable): variable(featureName=gCV_12_M)
  Set SingleDigitalPulseActionState SingleDigitalPulseActionState(hiPulseInSeconds=3, pin=GP_bool_out[17])
  MoveL speed 500 mm/s, acceleration 140 mm/s^2 (useActiveTCP=false) tcp=TCP_1; feature=CV
    Waypoint Variable (Variable): variable(featureName=gCV_13_M)
    Waypoint Variable (Variable): variable(featureName=gCV_14_M)
  SetPayload (workpieceName=k10)
SubProgram SUB_001 [hidden by the author, left out]
SubProgram SUB_103 [hidden by the author, left out]
SubProgram SUB_107 (keepSynchronizedWithDisk=true) programFile=/programs/GD/SUB_107.urp
  Folder FREE_DRIVE
    Script: freedrive_mode()
    SetPayload (workpieceName=k2)
    Set NoAction tcp=ZERO
    Wait Sleep waitTime=1
    Script: end_freedrive_mode()
  Folder CV_CORR_RZ
    If UseCVCorr
      Set NoAction tcp=TCP_1
      Script: sync()
      Script: CurrPos_p=get_actual_tcp_pose()
      CurrposAligned := p[0,0,0,0,0,0]
      CurrposAligned := GET_ALIGNED_TCP(CurrposAligned)
      Script: GET_CVCORR_VALUE(CurrposAligned)
SubProgram SUB_120 (keepSynchronizedWithDisk=true) programFile=/programs/GD/SUB_120.urp
  If GPBI_WorkExists (checkContinuously=true)
    Folder TRANSFER
      Script: set_tcp(CutOffTCP)
      MoveL speed 150 mm/s, acceleration 30 mm/s^2 (useActiveTCP=true) feature=Base
        SetPayload (workpieceName=k10)
        Waypoint Variable (Variable): variable(featureName=g2GD_pos1)
        Wait Sleep waitTime=0.5
  If ( not GPBI_WorkExists)
    SubPrgResult := 820
    Wait Sleep waitTime=999999
SubProgram SUB_161 [hidden by the author, left out]
SubProgram SUB_181 [hidden by the author, left out]
SubProgram SUB_141 (keepSynchronizedWithDisk=true) programFile=/programs/GD/SUB_141.urp
  Folder INITIALIZE
    SetPayload (workpieceName=k10)
    Script: pBucket[WorkPosNo]=p[0.,0.,0.,0.,0.,0.]
    If (WorkPosNo≟0)
      GD_pos4 := Capt_2BK_pos1
      GD_pos5 := Capt_2BK_pos2
      Capt_BK_L := Capt_2BK_L
      Capt_BK_R := Capt_2BK_R
    ElseIf (WorkPosNo≟1)
      GD_pos4 := Capt_1BK_pos1
      GD_pos5 := Capt_1BK_pos2
      Capt_BK_L := Capt_1BK_L
      Capt_BK_R := Capt_1BK_R
  Folder HOME
    SuppressedNode
      MoveJ speed 70 deg/s, acceleration 30 deg/s^2 (useActiveTCP=false) tcp=TCP_1; feature=Base
        Waypoint Variable (Variable): variable=GD_pos4
    SuppressedNode
      MoveL speed 200 mm/s, acceleration 70 mm/s^2 (useActiveTCP=true) feature=Base
        Waypoint Variable (Variable): variable=GD_pos5
  Folder ROVI_RECIPE
    If ( not ROVI_RECIPE(GPII_BucketNo))
      SubPrgResult := rovi_err
      Wait Sleep waitTime=999999
  Folder ROVI_RESET
    If ( not ROVI_RESET())
      SubPrgResult := rovi_err
      Wait Sleep waitTime=999999
  Folder ROVI_CAPTURE_1
    MoveL speed 250 mm/s, acceleration 140 mm/s^2 (useActiveTCP=false) tcp=TCP_1; feature=Base
      Waypoint Variable (Variable): variable(name=Capt_BK_L)
    Wait Sleep waitTime=1
    If ( not ROVI_CAPTURE())
      SubPrgResult := rovi_err
      Wait Sleep waitTime=999999
  Folder ROVI_CAPTURE_2
    MoveL speed 500 mm/s, acceleration 140 mm/s^2 (useActiveTCP=false) tcp=TCP_1; feature=Base
      Waypoint Variable (Variable): variable(name=Capt_BK_R)
    Wait Sleep waitTime=1
    If ( not ROVI_CAPTURE())
      SubPrgResult := rovi_err
      Wait Sleep waitTime=999999
  Folder ROVI_SOLVE
    Y2 := ROVI_SOLVE()
    If (Y2[0]≟10000.)
      SubPrgResult := rovi_err
      Wait Sleep waitTime=999999
  Folder ROVI_PARAM
    If not ROVI_PARAM(BKWidth_Name)
      SubPrgResult := rovi_err
      Wait Sleep waitTime=999999
    Script: BKWidth_Value[WorkPosNo]=Y8
  Folder HOME
    SuppressedNode
      MoveL speed 250 mm/s, acceleration 140 mm/s^2 (useActiveTCP=false) tcp=TCP_1; feature=Base
        Waypoint Variable (Variable): variable=GD_pos5
        Waypoint Variable (Variable): variable=GD_pos4
SubProgram SUB_143 (keepSynchronizedWithDisk=true) programFile=/programs/GD/SUB_143.urp
  Script: SET_BUCKET_DEF()
  Folder ROVI_RESET
    If (not ROVI_RESET())
      SubPrgResult := rovi_err
      Wait Sleep waitTime=999999
  Folder ROVI_CAPTURE_1
    BucketUpperPos := GET_BUCKET_UPPER(1)
    MoveL speed 250 mm/s, acceleration 140 mm/s^2 (useActiveTCP=false) tcp=TCP_1; feature=Bucket
      Waypoint Variable (Variable): variable=BucketUpperPos
    Wait Sleep waitTime=1
    If ( not ROVI_CAPTURE())
      SubPrgResult := rovi_err
      Wait Sleep waitTime=999999
  Folder ROVI_CAPTURE_2
    BucketUpperPos := GET_BUCKET_UPPER(2)
    MoveL speed 250 mm/s, acceleration 140 mm/s^2 (useActiveTCP=false) tcp=TCP_1; feature=Bucket
      Waypoint Variable (Variable): variable=BucketUpperPos
    Wait Sleep waitTime=1
    If ( not ROVI_CAPTURE())
      SubPrgResult := rovi_err
      Wait Sleep waitTime=999999
  Folder JUDGEMENT
    If (Y1[0]≟0)
      SubPrgResult := 990
      Wait Sleep waitTime=999999
    CrankDepth := (-1)*Y1[1]/1000.0
    CaptRowNo := 1+floor((CrankDepth-CrankDepthFull)/CaptStepZ)
    If (CaptRowNo<1)
      CaptRowNo := 1
    Set ExpressionOutput pin=GPIO_CaptRowNo; expression=CaptRowNo
SubProgram SUB_142 (keepSynchronizedWithDisk=true) programFile=/programs/GD/SUB_142.urp
  Folder INITIALIZE
    SetPayload (workpieceName=k10)
  Folder ROVI_RECIPE
    If ( not ROVI_RECIPE(GPII_ConveyorNo))
      SubPrgResult := rovi_err
      Wait Sleep waitTime=999999
  Folder ROVI_RESET
    If ( not ROVI_RESET())
      SubPrgResult := rovi_err
      Wait Sleep waitTime=999999
  Folder ROVI_CAPTURE
    MoveL speed 200 mm/s, acceleration 70 mm/s^2 (useActiveTCP=false) tcp=TCP_1; feature=Base
      Waypoint Variable (Variable): variable(featureName=Capt_CV_M)
    Wait Sleep waitTime=2
    If ( not ROVI_CAPTURE())
      SubPrgResult := rovi_err
      Wait Sleep waitTime=999999
  SuppressedNode
    Popup Message (haltProgram=false message=ok? inputType=Text)
  Folder ROVI_SOLVE
    Y2 := ROVI_SOLVE()
    If (Y2[0]≟10000.)
      SubPrgResult := rovi_err
      Wait Sleep waitTime=999999
SubProgram SUB_3100 (keepSynchronizedWithDisk=true) programFile=/programs/GD/SUB_3100.urp
  Loop Forever
    Sub3100_Option := Sub3100_GPII18
    If (Sub3100_Option≤14)
      'MOVE'
      If GPBI_PrgRun (checkContinuously=true)
        Set ExpressionOutput pin=GPBO_PrgRun; expression=True
        If GPBI_BLLoad1
          If (1≤Sub3100_Option and Sub3100_Option≤4)
            SetPayload (workpieceName=k10)
          ElseIf (5≤Sub3100_Option and Sub3100_Option≤6)
            SetPayload (workpieceName=k120)
          ElseIf (7≤Sub3100_Option and Sub3100_Option≤12)
            SetPayload (workpieceName=k10)
          ElseIf (13≤Sub3100_Option and Sub3100_Option≤14)
            SetPayload (workpieceName=k10)
        Else 
          If (1≤Sub3100_Option and Sub3100_Option≤4)
            SetPayload (workpieceName=k10)
          ElseIf (5≤Sub3100_Option and Sub3100_Option≤6)
            SetPayload (workpieceName=k120)
          ElseIf (7≤Sub3100_Option and Sub3100_Option≤12)
            SetPayload (workpieceName=k10)
          ElseIf (13≤Sub3100_Option and Sub3100_Option≤14)
            SetPayload (workpieceName=k10)
        Loop Forever
          Sub3100_Xd := [0.,0.,0.,0.,0.,0.]
          Sub3100_q := floor((Sub3100_Option-1) / 2)
          Sub3100_e := 1-((Sub3100_Option-1) % 2)*2
          Sub3100_t := 0.5
          If (1≤Sub3100_Option and Sub3100_Option≤6)
            '1:X+,2:X-,3:Y+,4:Y-,5:Z+,6:Z-'
            Script: Sub3100_Xd[Sub3100_q]=Sub3100_XdV*Sub3100_e
            If Sub3100_Option≟5
              If CurrPos[2]<Sub3100_ZMax (checkContinuously=true)
                Script: speedl(Sub3100_Xd,Sub3100_a,t=Sub3100_t)
              Script: stopl(Sub3100_d)
            Else 
              Script: speedl(Sub3100_Xd,Sub3100_a,t=Sub3100_t)
          ElseIf (7≤Sub3100_Option and Sub3100_Option≤12)
            '7:RX+,8:RX-,9:RY+,10:RY-,11:RZ+,12:RZ-'
            Script: Sub3100_Xd[Sub3100_q]=d2r(Sub3100_XdRot)*Sub3100_e
            Script: speedl(Sub3100_Xd,Sub3100_aRot,Sub3100_t)
          ElseIf (Sub3100_Option≟13 or Sub3100_Option≟14)
            '13:TZ+,14:TZ-'
            SuppressedNode
              Sub3100_curr := CurrPos_p
            Sub3100_curr := pose_trans(CurrPos, TCP3100TL)
            var_1 := p[0.,0.,0.,0.,0.,0.]
            Script: var_1[Sub3100_q-4]=0.25*Sub3100_e
            forceON := pose_sub(pose_trans(Sub3100_curr,var_1),Sub3100_curr)
            var_3 := 0
            Loop Counting (count=6) loopVariable(name=ループ_1)
              Script: Sub3100_Xd[var_3]=forceON[var_3]
              var_3 := var_3+1
            Script: speedl(Sub3100_Xd,Sub3100_a,Sub3100_t)
      Script: stopl(Sub3100_d)
    ElseIf (Sub3100_Option≤44)
      'FORCE'
      If GPBI_PrgRun
        Set ExpressionOutput pin=GPBO_PrgRun; expression=True
        If GPBI_BLLoad1
          If (33≤Sub3100_Option and Sub3100_Option≤36)
            SetPayload (workpieceName=k05)
          ElseIf (37≤Sub3100_Option and Sub3100_Option≤38)
            SetPayload (workpieceName=k05)
          ElseIf (39≤Sub3100_Option and Sub3100_Option≤44)
            SetPayload (workpieceName=k05)
        Else 
          If (33≤Sub3100_Option and Sub3100_Option≤36)
            SetPayload (workpieceName=k05)
          ElseIf (37≤Sub3100_Option and Sub3100_Option≤38)
            SetPayload (workpieceName=k05)
          ElseIf (39≤Sub3100_Option and Sub3100_Option≤44)
            SetPayload (workpieceName=k05)
        If (Sub3100_Option≟33)
          '33:X+'
          Force Frame feature=Base; selection=[1, 1, 1, 1, 1, 1]; wrench=[40, 0, 0, 0, 0, 0]; limitsForce=[0.01, 0.005, 0.005, 0.034907, 0.034907, 0.034907]; limitsMotion=[0.1, 0.1, 0.1, 0.349066, 0.349066, 0.349066]
            Wait DigitalInput pin=GPBI_PrgRun; digitalValue=0
        ElseIf (Sub3100_Option≟34)
          '34:X-'
          Force Frame feature=Base; selection=[1, 1, 1, 1, 1, 1]; wrench=[-40, 0, 0, 0, 0, 0]; limitsForce=[0.01, 0.005, 0.005, 0.034907, 0.034907, 0.034907]; limitsMotion=[0.1, 0.1, 0.1, 0.349066, 0.349066, 0.349066]
            Wait DigitalInput pin=GPBI_PrgRun; digitalValue=0
        ElseIf (Sub3100_Option≟35)
          '35:Y+'
          Force Frame feature=Base; selection=[1, 1, 1, 1, 1, 1]; wrench=[0, 40, 0, 0, 0, 0]; limitsForce=[0.005, 0.01, 0.005, 0.034907, 0.034907, 0.034907]; limitsMotion=[0.1, 0.1, 0.1, 0.349066, 0.349066, 0.349066]
            Wait DigitalInput pin=GPBI_PrgRun; digitalValue=0
        ElseIf (Sub3100_Option≟36)
          '36:Y-'
          Force Frame feature=Base; selection=[1, 1, 1, 1, 1, 1]; wrench=[0, -40, 0, 0, 0, 0]; limitsForce=[0.005, 0.01, 0.005, 0.034907, 0.034907, 0.034907]; limitsMotion=[0.1, 0.1, 0.1, 0.349066, 0.349066, 0.349066]
            Wait DigitalInput pin=GPBI_PrgRun; digitalValue=0
        ElseIf (Sub3100_Option≟37)
          '37:Z+'
          Force Frame feature=Base; selection=[1, 1, 1, 1, 1, 1]; wrench=[0, 0, 40, 0, 0, 0]; limitsForce=[0.005, 0.005, 0.01, 0.034907, 0.034907, 0.034907]; limitsMotion=[0.1, 0.1, 0.1, 0.349066, 0.349066, 0.349066]
            Wait DigitalInput pin=GPBI_PrgRun; digitalValue=0
        ElseIf (Sub3100_Option≟38)
          '38:Z-'
          Force Frame feature=Base; selection=[1, 1, 1, 1, 1, 1]; wrench=[0, 0, -40, 0, 0, 0]; limitsForce=[0.005, 0.005, 0.01, 0.034907, 0.034907, 0.034907]; limitsMotion=[0.1, 0.1, 0.1, 0.349066, 0.349066, 0.349066]
            Wait DigitalInput pin=GPBI_PrgRun; digitalValue=0
        ElseIf (Sub3100_Option≟39)
          '39:RX+'
          Force Frame feature=Base; selection=[1, 1, 1, 1, 1, 1]; wrench=[0, 0, 0, 40, 0, 0]; limitsForce=[0.005, 0.005, 0.005, 0.087266, 0.034907, 0.034907]; limitsMotion=[0.1, 0.1, 0.1, 0.349066, 0.349066, 0.349066]
            Wait DigitalInput pin=GPBI_PrgRun; digitalValue=0
        ElseIf (Sub3100_Option≟40)
          '40:RX-'
          Force Frame feature=Base; selection=[1, 1, 1, 1, 1, 1]; wrench=[0, 0, 0, -40, 0, 0]; limitsForce=[0.005, 0.005, 0.005, 0.087266, 0.034907, 0.034907]; limitsMotion=[0.1, 0.1, 0.1, 0.349066, 0.349066, 0.349066]
            Wait DigitalInput pin=GPBI_PrgRun; digitalValue=0
        ElseIf (Sub3100_Option≟41)
          '41:RY+'
          Force Frame feature=Base; selection=[1, 1, 1, 1, 1, 1]; wrench=[0, 0, 0, 0, 40, 0]; limitsForce=[0.005, 0.005, 0.005, 0.034907, 0.087266, 0.034907]; limitsMotion=[0.1, 0.1, 0.1, 0.349066, 0.349066, 0.349066]
            Wait DigitalInput pin=GPBI_PrgRun; digitalValue=0
        ElseIf (Sub3100_Option≟42)
          '42:RY-'
          Force Frame feature=Base; selection=[1, 1, 1, 1, 1, 1]; wrench=[0, 0, 0, 0, -40, 0]; limitsForce=[0.005, 0.005, 0.005, 0.034907, 0.087266, 0.034907]; limitsMotion=[0.1, 0.1, 0.1, 0.349066, 0.349066, 0.349066]
            Wait DigitalInput pin=GPBI_PrgRun; digitalValue=0
        ElseIf (Sub3100_Option≟43)
          '43:RZ+'
          Force Frame feature=Base; selection=[1, 1, 1, 1, 1, 1]; wrench=[0, 0, 0, 0, 0, 40]; limitsForce=[0.005, 0.005, 0.005, 0.034907, 0.034907, 0.087266]; limitsMotion=[0.1, 0.1, 0.1, 0.349066, 0.349066, 0.349066]
            Wait DigitalInput pin=GPBI_PrgRun; digitalValue=0
        ElseIf (Sub3100_Option≟44)
          '44:RZ-'
          Force Frame feature=Base; selection=[1, 1, 1, 1, 1, 1]; wrench=[0, 0, 0, 0, 0, -40]; limitsForce=[0.005, 0.005, 0.005, 0.034907, 0.034907, 0.087266]; limitsMotion=[0.1, 0.1, 0.1, 0.349066, 0.349066, 0.349066]
            Wait DigitalInput pin=GPBI_PrgRun; digitalValue=0
    ElseIf (Sub3100_Option≥90)
      'FREEDRIVE'
      If GPBI_PrgRun
        Set ExpressionOutput pin=GPBO_PrgRun; expression=True
        If GPBI_BLLoad1
          SetPayload (workpieceName=k05)
        Else 
          SetPayload (workpieceName=k05)
        If (Sub3100_Option≟90)
          '90:FreeDrive'
          Script: freedrive_mode()
          Wait DigitalInput pin=GPBI_PrgRun; digitalValue=0
          Script: end_freedrive_mode()
    Script: stopl(Sub3100_d)
    Wait Sleep waitTime=0.01
    SetPayload (workpieceName=k10)
    Set ExpressionOutput pin=GPBO_PrgRun; expression=False
SubProgram SUB_6001 (keepSynchronizedWithDisk=true) programFile=/programs/GD/SUB_6001.urp
  SetPayload (workpieceName=k10)
  If ( not ROVI_RESET())
    SubPrgResult := rovi_err
    Wait Sleep waitTime=999999
  MoveJ speed 9 deg/s, acceleration 15 deg/s^2 (useActiveTCP=false) tcp=ZERO; feature=Base
    Waypoint CaptPos0: TCP in base x=893.15 y=-272.89 z=528.478 mm, rx=-2.1539 ry=2.287 rz=-0.0001 rad; joints [-6.349, -112.609, -77.746, -79.721, 90.331, -2.756] deg
  CaptPos := CaptPos0_p
  Loop While (checkContinuously=false) expression=(CaptPos[0]≠10000.0)
    MoveJ speed 9 deg/s, acceleration 15 deg/s^2 (useActiveTCP=false) tcp=ZERO; feature=Base
      Waypoint Variable (Variable): variable=CaptPos
    Wait Sleep waitTime=4
    If ( not ROVI_CAPTURE())
      SubPrgResult := rovi_err
      Wait Sleep waitTime=999999
    CaptPos := ROVI_SOLVE(is_popup=False)
  MoveJ speed 9 deg/s, acceleration 15 deg/s^2 (useActiveTCP=false) tcp=ZERO; feature=Base
    Waypoint CaptPos0: TCP in base x=893.15 y=-272.89 z=528.478 mm, rx=-2.1539 ry=2.287 rz=-0.0001 rad; joints [-6.349, -112.609, -77.746, -79.721, 90.331, -2.756] deg
SubProgram SUB_6101 (keepSynchronizedWithDisk=true) programFile=/programs/GD/SUB_6101.urp
  Folder ROVI_RECIPE
    If (not ROVI_RECIPE(GPII_WorkNo))
      SubPrgResult := rovi_err
      Wait Sleep waitTime=999999
  Folder ROVI_RESET
    If ( not ROVI_RESET())
      SubPrgResult := rovi_err
      Wait Sleep waitTime=999999
  Folder ROVI_CAPTURE_1
    MoveJ speed 6 deg/s, acceleration 12 deg/s^2 (useActiveTCP=false) tcp=TCP_1; feature=Base
      Switch expression=CheckMST
        Case (caseValue=0)
          Waypoint Variable (Variable): variable(featureName=Master_pos)
        Case (caseValue=1)
          Waypoint Variable (Variable): variable(featureName=Master_pos)
        Case (caseValue=2)
          Waypoint Variable (Variable): variable(featureName=Master_posL)
        Case (caseValue=3)
          Waypoint Variable (Variable): variable(featureName=Master_posR)
      SuppressedNode
        Waypoint ウェイポイント_1 (Relative): relativeFromPosition TCP in base x=-5.037 y=-329.575 z=16.043 mm, rx=-0.0235 ry=-3.1385 rz=-0.002 rad; joints [-65.945, -61.292, -135.715, -73.119, 89.887, 25.023] deg; TCP offset x=0 y=80 z=420 mm, rx=0 ry=0 rz=0 rad; TCP in base x=-3.24 y=-405.091 z=93.349 mm, rx=0.0238 ry=2.9687 rz=0.0105 rad; joints [-81.058, -70.218, -123.998, -74.522, 99.793, 10.078] deg
    Wait Sleep waitTime=3
    If ( not ROVI_CAPTURE())
      SubPrgResult := rovi_err
      Wait Sleep waitTime=999999
SubProgram SUB_6102 [hidden by the author, left out]
SubProgram SUB_6102RX [hidden by the author, left out]
SubProgram SUB_6102RXF [hidden by the author, left out]
SubProgram SUB_6102RXFF (keepSynchronizedWithDisk=true) programFile=/programs/GD/SUB_6102RXFF.urp
  SetPayload (workpieceName=k10)
  UF := Base
  If (GPII_CheckMST>0)
    Folder ROVI_SOLVE
      If (CandCnt>0)
        Y2 := ROVI_SOLVE()
        If (Y2[0]≟10000.)
          SubPrgResult := rovi_err
          Wait Sleep waitTime=999999
    UF := Y2
  Folder M
    MoveL speed 120 mm/s, acceleration 70 mm/s^2 (useActiveTCP=false) tcp=TCP_RX; feature=UF
      Waypoint Variable (Variable): variable(featureName=gGD_3_M_RX)
      Wait Sleep waitTime=1
      Waypoint Variable (Variable): variable(featureName=gGD_2_M_RX)
      Wait Sleep waitTime=1
      Set SingleDigitalPulseActionState SingleDigitalPulseActionState(hiPulseInSeconds=1, pin=GP_bool_out[14])
      Popup Message (haltProgram=false message=ok? inputType=Text)
    Timer (action=Reset) variable(name=tm_6102_01)
    Timer (action=Start) variable=tm_6102_01
    SuppressedNode
      Force Frame feature=Joint_6_name; selection=[1, 1, 1, 0, 0, 0]; wrench=[0, 0, 10, 0, 0, 0]; limitsForce=[0.005, 0.005, 0.04, 0.034907, 0.034907, 1.047198]; limitsMotion=[0.1, 0.1, 0.1, 0.349066, 0.349066, 0.349066]
        ShakeCnt := -1
        Loop While (checkContinuously=false) expression=((Currpos_p_UF0[1]>(gGD_2_M_RX[1]-HandInZ)) and (tm_6102_01<GPII_TMHandIn))
          IsShake := False
          If ShakeCnt<0
            Folder NOT_SHAKE
              Timer (action=Start) variable(name=tm_6102_02)
              Wait Condition expression=tm_6102_02>ShakeWaitSec
              Timer (action=Stop) variable=tm_6102_02
              Timer (action=Reset) variable=tm_6102_02
            ShakeCnt := 0
          Folder MONITOR_SPEED
            Timer (action=Reset) variable=tm_6102_02
            If norm(TCPSpeed[2])<TCPSpeedThZ
              IsShake := True
              If ShakeCnt≟0
                Timer (action=Start) variable=tm_6102_02
                Loop While (checkContinuously=false) expression=((tm_6102_02<1.0) and (IsShake≟ True ))
                  If norm(TCPSpeed[2])≥TCPSpeedThZ
                    IsShake := False
                Timer (action=Stop) variable=tm_6102_02
              ShakeCnt := ShakeCnt+1
          Folder SHAKE
            If IsShake
              Sub3100_Option := 9
              Loop Counting (count=2) loopVariable(name=ループ_6)
                '7:RX+,8:RX-,9:RY+,10:RY-,11:RZ+,12:RZ-'
                Sub3100_Xd := [0.,0.,0.,0.,0.,0.]
                Sub3100_q := floor((Sub3100_Option-1) / 2)
                Sub3100_e := 1-((Sub3100_Option-1) % 2)*2
                Sub3100_t := 0.2
                Script: Sub3100_Xd[Sub3100_q]=d2r(Sub3100_XdRot/2.0)*Sub3100_e
                Script: speedl(Sub3100_Xd,Sub3100_aRot/2.0,Sub3100_t)
                If Sub3100_Option≟9
                  Sub3100_Option := 10
                Else 
                  Sub3100_Option := 9
